   DATA[1964,13] := 797.9124;
   DATA[1964,14] := 1.0;
   DATA[1964,15] := 2.0;
   DATA[1964,16] := 1.0;
   DATA[1964,17] := 1.0;
   DATA[1964,18] := 1.0;
   DATA[1964,19] := 2.0;
   DATA[1964,20] := 148.808;
   DATA[1964,21] := 154.8065;
   DATA[1964,22] := 1.718387;
   DATA[1964,23] := 826.5958;
   DATA[1964,24] := 2.0;
   DATA[1964,25] := 2.0;
   DATA[1964,26] := 7.874455;
   DATA[1964,27] := 143.8093;
   DATA[1964,28] := 262.2084;
   DATA[1964,29] := 12.11228;
   DATA[1964,30] := 1.72725;
   DATA[1964,31] := 1.264891;
   DATA[1964,32] := 0.7352687;
   DATA[1964,33] := 0.3079781;
   DATA[1964,34] := 2.0;
   DATA[1964,35] := 250.5768;
   DATA[1964,36] := 1.730048;
   DATA[1964,37] := 189.3265;
   DATA[1964,38] := 0.000128152;
   DATA[1964,39] := 1.0;
   DATA[1964,40] := 1.0;
   DATA[1965,0] := 2.537873;
   DATA[1965,1] := 860.8522;
   DATA[1965,2] := 2.0;
   DATA[1965,3] := 2.0;
   DATA[1965,4] := 262.3686;
   DATA[1965,5] := 8.396437;
   DATA[1965,6] := 331.8893;
   DATA[1965,7] := 2.462051;
   DATA[1965,8] := 2.0;
   DATA[1965,9] := 2.0;
   DATA[1965,10] := 2.0;
   DATA[1965,11] := 19.69396;
   DATA[1965,12] := 2.209269;
   DATA[1965,13] := 797.8724;
   DATA[1965,14] := 1.0;
   DATA[1965,15] := 2.0;
   DATA[1965,16] := 1.0;
   DATA[1965,17] := 1.0;
   DATA[1965,18] := 1.0;
   DATA[1965,19] := 2.0;
   DATA[1965,20] := 148.808;
   DATA[1965,21] := 154.8065;
   DATA[1965,22] := 1.718771;
   DATA[1965,23] := 826.5189;
   DATA[1965,24] := 2.0;
   DATA[1965,25] := 2.0;
   DATA[1965,26] := 7.874455;
   DATA[1965,27] := 143.8093;
   DATA[1965,28] := 262.2084;
   DATA[1965,29] := 12.11228;
   DATA[1965,30] := 1.72725;
   DATA[1965,31] := 1.262073;
   DATA[1965,32] := 0.7352687;
   DATA[1965,33] := 0.3079781;
   DATA[1965,34] := 2.0;
   DATA[1965,35] := 250.5768;
   DATA[1965,36] := 1.730048;
   DATA[1965,37] := 189.3265;
   DATA[1965,38] := 0.000128152;
   DATA[1965,39] := 1.0;
   DATA[1965,40] := 1.0;
   DATA[1966,0] := 2.58111;
   DATA[1966,1] := 860.6559;
   DATA[1966,2] := 2.0;
   DATA[1966,3] := 2.0;
   DATA[1966,4] := 262.3686;
   DATA[1966,5] := 8.396437;
   DATA[1966,6] := 331.8893;
   DATA[1966,7] := 2.46077;
   DATA[1966,8] := 2.0;
   DATA[1966,9] := 2.0;
   DATA[1966,10] := 2.0;
   DATA[1966,11] := 19.74838;
   DATA[1966,12] := 2.21119;
   DATA[1966,13] := 797.7522;
   DATA[1966,14] := 1.0;
   DATA[1966,15] := 2.0;
   DATA[1966,16] := 1.0;
   DATA[1966,17] := 1.0;
   DATA[1966,18] := 1.0;
   DATA[1966,19] := 2.0;
   DATA[1966,20] := 148.808;
   DATA[1966,21] := 154.8065;
   DATA[1966,22] := 1.720437;
   DATA[1966,23] := 826.1728;
   DATA[1966,24] := 2.0;
   DATA[1966,25] := 2.0;
   DATA[1966,26] := 7.874455;
   DATA[1966,27] := 143.8349;
   DATA[1966,28] := 262.2084;
   DATA[1966,29] := 12.11228;
   DATA[1966,30] := 1.72725;
   DATA[1966,31] := 1.276162;
   DATA[1966,32] := 0.7352687;
   DATA[1966,33] := 0.3084905;
   DATA[1966,34] := 2.0;
   DATA[1966,35] := 250.5768;
   DATA[1966,36] := 1.730048;
   DATA[1966,37] := 189.3265;
   DATA[1966,38] := 0.000128152;
   DATA[1966,39] := 1.0;
   DATA[1966,40] := 1.0;
   DATA[1967,0] := 2.61602;
   DATA[1967,1] := 860.6167;
   DATA[1967,2] := 2.0;
   DATA[1967,3] := 2.0;
   DATA[1967,4] := 262.3686;
   DATA[1967,5] := 8.396437;
   DATA[1967,6] := 331.8893;
   DATA[1967,7] := 2.46077;
   DATA[1967,8] := 2.0;
   DATA[1967,9] := 2.0;
   DATA[1967,10] := 2.0;
   DATA[1967,11] := 19.79;
   DATA[1967,12] := 2.212343;
   DATA[1967,13] := 797.5119;
   DATA[1967,14] := 1.0;
   DATA[1967,15] := 2.0;
   DATA[1967,16] := 1.0;
   DATA[1967,17] := 1.0;
   DATA[1967,18] := 1.0;
   DATA[1967,19] := 2.0;
   DATA[1967,20] := 148.808;
   DATA[1967,21] := 154.8065;
   DATA[1967,22] := 1.721206;
   DATA[1967,23] := 826.3651;
   DATA[1967,24] := 2.0;
   DATA[1967,25] := 2.0;
   DATA[1967,26] := 7.874455;
   DATA[1967,27] := 144.0144;
   DATA[1967,28] := 262.2084;
   DATA[1967,29] := 12.11228;
   DATA[1967,30] := 1.72725;
   DATA[1967,31] := 1.289996;
   DATA[1967,32] := 0.7352687;
   DATA[1967,33] := 0.3086186;
   DATA[1967,34] := 2.0;
   DATA[1967,35] := 250.5768;
   DATA[1967,36] := 1.730048;
   DATA[1967,37] := 189.3265;
   DATA[1967,38] := 0.000128152;
   DATA[1967,39] := 1.0;
   DATA[1967,40] := 1.0;
   DATA[1968,0] := 2.6394;
   DATA[1968,1] := 860.9307;
   DATA[1968,2] := 2.0;
   DATA[1968,3] := 2.0;
   DATA[1968,4] := 262.3686;
   DATA[1968,5] := 8.396437;
   DATA[1968,6] := 331.8123;
   DATA[1968,7] := 2.46077;
   DATA[1968,8] := 2.0;
   DATA[1968,9] := 2.0;
   DATA[1968,10] := 2.0;
   DATA[1968,11] := 19.79;
   DATA[1968,12] := 2.212343;
   DATA[1968,13] := 797.7922;
   DATA[1968,14] := 1.0;
   DATA[1968,15] := 2.0;
   DATA[1968,16] := 1.0;
   DATA[1968,17] := 1.0;
   DATA[1968,18] := 1.0;
   DATA[1968,19] := 2.0;
   DATA[1968,20] := 148.808;
   DATA[1968,21] := 154.8065;
   DATA[1968,22] := 1.721206;
   DATA[1968,23] := 825.9805;
   DATA[1968,24] := 2.0;
   DATA[1968,25] := 2.0;
   DATA[1968,26] := 7.874455;
   DATA[1968,27] := 144.0144;
   DATA[1968,28] := 262.2084;
   DATA[1968,29] := 12.11228;
   DATA[1968,30] := 1.72725;
   DATA[1968,31] := 1.302933;
   DATA[1968,32] := 0.7352687;
   DATA[1968,33] := 0.3086186;
   DATA[1968,34] := 2.0;
   DATA[1968,35] := 250.5768;
   DATA[1968,36] := 1.730048;
   DATA[1968,37] := 189.3265;
   DATA[1968,38] := 0.000128152;
   DATA[1968,39] := 1.0;
   DATA[1968,40] := 1.0;
   DATA[1969,0] := 2.652532;
   DATA[1969,1] := 860.9307;
   DATA[1969,2] := 2.0;
   DATA[1969,3] := 2.0;
   DATA[1969,4] := 262.3686;
   DATA[1969,5] := 8.396437;
   DATA[1969,6] := 331.8123;
   DATA[1969,7] := 2.46077;
   DATA[1969,8] := 2.0;
   DATA[1969,9] := 2.0;
   DATA[1969,10] := 2.0;
   DATA[1969,11] := 19.79;
   DATA[1969,12] := 2.21055;
   DATA[1969,13] := 797.592;
   DATA[1969,14] := 1.0;
   DATA[1969,15] := 2.0;
   DATA[1969,16] := 1.0;
   DATA[1969,17] := 1.0;
   DATA[1969,18] := 1.0;
   DATA[1969,19] := 2.0;
   DATA[1969,20] := 148.808;
   DATA[1969,21] := 154.8065;
   DATA[1969,22] := 1.720437;
   DATA[1969,23] := 825.6345;
   DATA[1969,24] := 2.0;
   DATA[1969,25] := 2.0;
   DATA[1969,26] := 7.874455;
   DATA[1969,27] := 144.0144;
   DATA[1969,28] := 262.2084;
   DATA[1969,29] := 12.11228;
   DATA[1969,30] := 1.72725;
   DATA[1969,31] := 1.310106;
   DATA[1969,32] := 0.7352687;
   DATA[1969,33] := 0.3072735;
   DATA[1969,34] := 2.0;
   DATA[1969,35] := 250.5768;
   DATA[1969,36] := 1.730048;
   DATA[1969,37] := 189.3265;
   DATA[1969,38] := 0.000128152;
   DATA[1969,39] := 1.0;
   DATA[1969,40] := 1.0;
   DATA[1970,0] := 2.656375;
   DATA[1970,1] := 860.5382;
   DATA[1970,2] := 2.0;
   DATA[1970,3] := 2.0;
   DATA[1970,4] := 262.3686;
   DATA[1970,5] := 8.396437;
   DATA[1970,6] := 331.8123;
   DATA[1970,7] := 2.46077;
   DATA[1970,8] := 2.0;
   DATA[1970,9] := 2.0;
   DATA[1970,10] := 2.0;
   DATA[1970,11] := 19.75479;
   DATA[1970,12] := 2.209269;
   DATA[1970,13] := 797.7522;
   DATA[1970,14] := 1.0;
   DATA[1970,15] := 2.0;
   DATA[1970,16] := 1.0;
   DATA[1970,17] := 1.0;
   DATA[1970,18] := 1.0;
   DATA[1970,19] := 2.0;
   DATA[1970,20] := 148.808;
   DATA[1970,21] := 154.8065;
   DATA[1970,22] := 1.720437;
   DATA[1970,23] := 825.596;
   DATA[1970,24] := 2.0;
   DATA[1970,25] := 2.0;
   DATA[1970,26] := 7.874455;
   DATA[1970,27] := 143.8862;
   DATA[1970,28] := 262.2084;
   DATA[1970,29] := 12.11228;
   DATA[1970,30] := 1.72725;
   DATA[1970,31] := 1.302293;
   DATA[1970,32] := 0.7352687;
   DATA[1970,33] := 0.3069532;
   DATA[1970,34] := 2.0;
   DATA[1970,35] := 250.5768;
   DATA[1970,36] := 1.730048;
   DATA[1970,37] := 189.4226;
   DATA[1970,38] := 0.000128152;
   DATA[1970,39] := 1.0;
   DATA[1970,40] := 1.0;
   DATA[1971,0] := 2.639721;
   DATA[1971,1] := 860.2242;
   DATA[1971,2] := 2.0;
   DATA[1971,3] := 2.0;
   DATA[1971,4] := 262.3686;
   DATA[1971,5] := 8.396437;
   DATA[1971,6] := 331.6842;
   DATA[1971,7] := 2.461539;
   DATA[1971,8] := 2.0;
   DATA[1971,9] := 2.0;
   DATA[1971,10] := 2.0;
   DATA[1971,11] := 19.75479;
   DATA[1971,12] := 2.209013;
   DATA[1971,13] := 797.7922;
   DATA[1971,14] := 1.0;
   DATA[1971,15] := 2.0;
   DATA[1971,16] := 1.0;
   DATA[1971,17] := 1.0;
   DATA[1971,18] := 1.0;
   DATA[1971,19] := 2.0;
   DATA[1971,20] := 148.808;
   DATA[1971,21] := 154.8065;
   DATA[1971,22] := 1.720437;
   DATA[1971,23] := 826.019;
   DATA[1971,24] := 2.0;
   DATA[1971,25] := 2.0;
   DATA[1971,26] := 7.874455;
   DATA[1971,27] := 143.8862;
   DATA[1971,28] := 262.2084;
   DATA[1971,29] := 12.11228;
   DATA[1971,30] := 1.729172;
   DATA[1971,31] := 1.292814;
   DATA[1971,32] := 0.7352687;
   DATA[1971,33] := 0.3069532;
   DATA[1971,34] := 2.0;
   DATA[1971,35] := 250.5768;
   DATA[1971,36] := 1.730048;
   DATA[1971,37] := 189.4226;
   DATA[1971,38] := 0.000128152;
   DATA[1971,39] := 1.0;
   DATA[1971,40] := 1.0;
   DATA[1972,0] := 2.626909;
   DATA[1972,1] := 860.1064;
   DATA[1972,2] := 2.0;
   DATA[1972,3] := 2.0;
   DATA[1972,4] := 262.3686;
   DATA[1972,5] := 8.396437;
   DATA[1972,6] := 331.6842;
   DATA[1972,7] := 2.462564;
   DATA[1972,8] := 2.0;
   DATA[1972,9] := 2.0;
   DATA[1972,10] := 2.0;
   DATA[1972,11] := 19.71957;
   DATA[1972,12] := 2.209013;
   DATA[1972,13] := 797.6721;
   DATA[1972,14] := 1.0;
   DATA[1972,15] := 2.0;
   DATA[1972,16] := 1.0;
   DATA[1972,17] := 1.0;
   DATA[1972,18] := 1.0;
   DATA[1972,19] := 2.0;
   DATA[1972,20] := 148.808;
   DATA[1972,21] := 154.8065;
   DATA[1972,22] := 1.719796;
   DATA[1972,23] := 825.7883;
   DATA[1972,24] := 2.0;
   DATA[1972,25] := 2.0;
   DATA[1972,26] := 7.874455;
   DATA[1972,27] := 143.8862;
   DATA[1972,28] := 262.2084;
   DATA[1972,29] := 12.11228;
   DATA[1972,30] := 1.730197;
   DATA[1972,31] := 1.277956;
   DATA[1972,32] := 0.7352687;
   DATA[1972,33] := 0.3069532;
   DATA[1972,34] := 2.0;
   DATA[1972,35] := 250.5768;
   DATA[1972,36] := 1.730048;
   DATA[1972,37] := 189.4226;
   DATA[1972,38] := 0.000128152;
   DATA[1972,39] := 1.0;
   DATA[1972,40] := 1.0;
   DATA[1973,0] := 2.620184;
   DATA[1973,1] := 860.1457;
   DATA[1973,2] := 2.0;
   DATA[1973,3] := 2.0;
   DATA[1973,4] := 262.3686;
   DATA[1973,5] := 8.396437;
   DATA[1973,6] := 331.6842;
   DATA[1973,7] := 2.462564;
   DATA[1973,8] := 2.0;
   DATA[1973,9] := 2.0;
   DATA[1973,10] := 2.0;
   DATA[1973,11] := 19.70677;
   DATA[1973,12] := 2.209013;
   DATA[1973,13] := 797.6721;
   DATA[1973,14] := 1.0;
   DATA[1973,15] := 2.0;
   DATA[1973,16] := 1.0;
   DATA[1973,17] := 1.0;
   DATA[1973,18] := 1.0;
   DATA[1973,19] := 2.0;
   DATA[1973,20] := 148.808;
   DATA[1973,21] := 154.8065;
   DATA[1973,22] := 1.719796;
   DATA[1973,23] := 825.9421;
   DATA[1973,24] := 2.0;
   DATA[1973,25] := 2.0;
   DATA[1973,26] := 7.874455;
   DATA[1973,27] := 143.8862;
   DATA[1973,28] := 262.2084;
   DATA[1973,29] := 12.11228;
   DATA[1973,30] := 1.731864;
   DATA[1973,31] := 1.272192;
   DATA[1973,32] := 0.7352687;
   DATA[1973,33] := 0.3069532;
   DATA[1973,34] := 2.0;
   DATA[1973,35] := 250.5127;
   DATA[1973,36] := 1.730048;
   DATA[1973,37] := 189.4226;
   DATA[1973,38] := 0.000128152;
   DATA[1973,39] := 1.0;
   DATA[1973,40] := 1.0;
   DATA[1974,0] := 2.613778;
   DATA[1974,1] := 859.9494;
   DATA[1974,2] := 2.0;
   DATA[1974,3] := 2.0;
   DATA[1974,4] := 262.3686;
   DATA[1974,5] := 8.396437;
   DATA[1974,6] := 331.6842;
   DATA[1974,7] := 2.462564;
   DATA[1974,8] := 2.0;
   DATA[1974,9] := 2.0;
   DATA[1974,10] := 2.0;
   DATA[1974,11] := 19.68436;
   DATA[1974,12] := 2.209525;
   DATA[1974,13] := 797.7522;
   DATA[1974,14] := 1.0;
   DATA[1974,15] := 2.0;
   DATA[1974,16] := 1.0;
   DATA[1974,17] := 1.0;
   DATA[1974,18] := 1.0;
   DATA[1974,19] := 2.0;
   DATA[1974,20] := 148.808;
   DATA[1974,21] := 154.8065;
   DATA[1974,22] := 1.71813;
   DATA[1974,23] := 826.1343;
   DATA[1974,24] := 2.0;
   DATA[1974,25] := 2.0;
   DATA[1974,26] := 7.874455;
   DATA[1974,27] := 143.8862;
   DATA[1974,28] := 262.2084;
   DATA[1974,29] := 12.11228;
   DATA[1974,30] := 1.731864;
   DATA[1974,31] := 1.265147;
   DATA[1974,32] := 0.7352687;
   DATA[1974,33] := 0.3069532;
   DATA[1974,34] := 2.0;
   DATA[1974,35] := 250.5127;
   DATA[1974,36] := 1.730048;
   DATA[1974,37] := 189.4226;
   DATA[1974,38] := 0.000128152;
   DATA[1974,39] := 1.0;
   DATA[1974,40] := 1.0;
   DATA[1975,0] := 2.601608;
   DATA[1975,1] := 859.8709;
   DATA[1975,2] := 2.0;
   DATA[1975,3] := 2.0;
   DATA[1975,4] := 262.3686;
   DATA[1975,5] := 8.396437;
   DATA[1975,6] := 331.6842;
   DATA[1975,7] := 2.462564;
   DATA[1975,8] := 2.0;
   DATA[1975,9] := 2.0;
   DATA[1975,10] := 2.0;
   DATA[1975,11] := 19.66195;
   DATA[1975,12] := 2.209525;
   DATA[1975,13] := 797.9925;
   DATA[1975,14] := 1.0;
   DATA[1975,15] := 2.0;
   DATA[1975,16] := 1.0;
   DATA[1975,17] := 1.0;
   DATA[1975,18] := 1.0;
   DATA[1975,19] := 2.0;
   DATA[1975,20] := 148.808;
   DATA[1975,21] := 154.8065;
   DATA[1975,22] := 1.71813;
   DATA[1975,23] := 826.442;
   DATA[1975,24] := 2.0;
   DATA[1975,25] := 2.0;
   DATA[1975,26] := 7.874455;
   DATA[1975,27] := 143.8862;
   DATA[1975,28] := 262.2084;
   DATA[1975,29] := 12.11228;
   DATA[1975,30] := 1.731095;
   DATA[1975,31] := 1.26425;
   DATA[1975,32] := 0.7352687;
   DATA[1975,33] := 0.3066329;
   DATA[1975,34] := 2.0;
   DATA[1975,35] := 250.5127;
   DATA[1975,36] := 1.730048;
   DATA[1975,37] := 189.4226;
   DATA[1975,38] := 0.000128152;
   DATA[1975,39] := 1.0;
   DATA[1975,40] := 1.0;
   DATA[1976,0] := 2.583352;
   DATA[1976,1] := 859.7139;
   DATA[1976,2] := 2.0;
   DATA[1976,3] := 2.0;
   DATA[1976,4] := 262.3686;
   DATA[1976,5] := 8.396437;
   DATA[1976,6] := 331.6842;
   DATA[1976,7] := 2.462564;
   DATA[1976,8] := 2.0;
   DATA[1976,9] := 2.0;
   DATA[1976,10] := 2.0;
   DATA[1976,11] := 19.66195;
   DATA[1976,12] := 2.209525;
   DATA[1976,13] := 797.9925;
   DATA[1976,14] := 1.0;
   DATA[1976,15] := 2.0;
   DATA[1976,16] := 1.0;
   DATA[1976,17] := 1.0;
   DATA[1976,18] := 1.0;
   DATA[1976,19] := 2.0;
   DATA[1976,20] := 148.808;
   DATA[1976,21] := 154.8065;
   DATA[1976,22] := 1.71813;
   DATA[1976,23] := 826.5189;
   DATA[1976,24] := 2.0;
   DATA[1976,25] := 2.0;
   DATA[1976,26] := 7.874455;
   DATA[1976,27] := 143.8862;
   DATA[1976,28] := 262.2084;
   DATA[1976,29] := 12.03538;
   DATA[1976,30] := 1.731095;
   DATA[1976,31] := 1.271935;
   DATA[1976,32] := 0.7352687;
   DATA[1976,33] := 0.3065048;
   DATA[1976,34] := 2.0;
   DATA[1976,35] := 250.5127;
   DATA[1976,36] := 1.730048;
   DATA[1976,37] := 189.4226;
   DATA[1976,38] := 0.000128152;
   DATA[1976,39] := 1.0;
   DATA[1976,40] := 1.0;
   DATA[1977,0] := 2.572463;
   DATA[1977,1] := 859.8317;
   DATA[1977,2] := 2.0;
   DATA[1977,3] := 2.0;
   DATA[1977,4] := 262.3686;
   DATA[1977,5] := 8.396437;
   DATA[1977,6] := 331.6842;
   DATA[1977,7] := 2.462564;
   DATA[1977,8] := 2.0;
   DATA[1977,9] := 2.0;
   DATA[1977,10] := 2.0;
   DATA[1977,11] := 19.70037;
   DATA[1977,12] := 2.209525;
   DATA[1977,13] := 798.353;
   DATA[1977,14] := 1.0;
   DATA[1977,15] := 2.0;
   DATA[1977,16] := 1.0;
   DATA[1977,17] := 1.0;
   DATA[1977,18] := 1.0;
   DATA[1977,19] := 2.0;
   DATA[1977,20] := 148.808;
   DATA[1977,21] := 154.8065;
   DATA[1977,22] := 1.71813;
   DATA[1977,23] := 826.5573;
   DATA[1977,24] := 2.0;
   DATA[1977,25] := 2.0;
   DATA[1977,26] := 7.874455;
   DATA[1977,27] := 143.8862;
   DATA[1977,28] := 262.2084;
   DATA[1977,29] := 12.03538;
   DATA[1977,30] := 1.731095;
   DATA[1977,31] := 1.271935;
   DATA[1977,32] := 0.7352687;
   DATA[1977,33] := 0.3065048;
   DATA[1977,34] := 2.0;
   DATA[1977,35] := 250.5127;
   DATA[1977,36] := 1.730048;
   DATA[1977,37] := 189.2464;
   DATA[1977,38] := 0.000128152;
   DATA[1977,39] := 1.0;
   DATA[1977,40] := 1.0;
   DATA[1978,0] := 2.556769;
   DATA[1978,1] := 859.6354;
   DATA[1978,2] := 2.0;
   DATA[1978,3] := 2.0;
   DATA[1978,4] := 262.3686;
   DATA[1978,5] := 8.396437;
   DATA[1978,6] := 331.6842;
   DATA[1978,7] := 2.462564;
   DATA[1978,8] := 2.0;
   DATA[1978,9] := 2.0;
   DATA[1978,10] := 2.0;
   DATA[1978,11] := 19.76439;
   DATA[1978,12] := 2.209525;
   DATA[1978,13] := 798.7535;
   DATA[1978,14] := 1.0;
   DATA[1978,15] := 2.0;
   DATA[1978,16] := 1.0;
   DATA[1978,17] := 1.0;
   DATA[1978,18] := 1.0;
   DATA[1978,19] := 2.0;
   DATA[1978,20] := 148.808;
   DATA[1978,21] := 154.8065;
   DATA[1978,22] := 1.716721;
   DATA[1978,23] := 826.6342;
   DATA[1978,24] := 2.0;
   DATA[1978,25] := 2.0;
   DATA[1978,26] := 7.874455;
   DATA[1978,27] := 143.8862;
   DATA[1978,28] := 262.2084;
   DATA[1978,29] := 12.03538;
   DATA[1978,30] := 1.7293;
   DATA[1978,31] := 1.280517;
   DATA[1978,32] := 0.7352687;
   DATA[1978,33] := 0.3065048;
   DATA[1978,34] := 2.0;
   DATA[1978,35] := 250.5127;
   DATA[1978,36] := 1.730048;
   DATA[1978,37] := 189.2464;
   DATA[1978,38] := 0.000128152;
   DATA[1978,39] := 1.0;
   DATA[1978,40] := 1.0;
   DATA[1979,0] := 2.53435;
   DATA[1979,1] := 859.9494;
   DATA[1979,2] := 2.0;
   DATA[1979,3] := 2.0;
   DATA[1979,4] := 262.3686;
   DATA[1979,5] := 8.396437;
   DATA[1979,6] := 331.6842;
   DATA[1979,7] := 2.462564;
   DATA[1979,8] := 2.0;
   DATA[1979,9] := 2.0;
   DATA[1979,10] := 2.0;
   DATA[1979,11] := 19.76439;
   DATA[1979,12] := 2.209525;
   DATA[1979,13] := 798.6735;
   DATA[1979,14] := 1.0;
   DATA[1979,15] := 2.0;
   DATA[1979,16] := 1.0;
   DATA[1979,17] := 1.0;
   DATA[1979,18] := 1.0;
   DATA[1979,19] := 2.0;
   DATA[1979,20] := 148.808;
   DATA[1979,21] := 154.8065;
   DATA[1979,22] := 1.716721;
   DATA[1979,23] := 826.3266;
   DATA[1979,24] := 2.0;
   DATA[1979,25] := 2.0;
   DATA[1979,26] := 7.874455;
   DATA[1979,27] := 143.8862;
   DATA[1979,28] := 262.2084;
   DATA[1979,29] := 12.03538;
   DATA[1979,30] := 1.728147;
   DATA[1979,31] := 1.280902;
   DATA[1979,32] := 0.7352687;
   DATA[1979,33] := 0.3065048;
   DATA[1979,34] := 2.0;
   DATA[1979,35] := 250.5127;
   DATA[1979,36] := 1.730048;
   DATA[1979,37] := 189.2464;
   DATA[1979,38] := 0.000128152;
   DATA[1979,39] := 1.0;
   DATA[1979,40] := 1.0;
   DATA[1980,0] := 2.518015;
   DATA[1980,1] := 859.6354;
   DATA[1980,2] := 2.0;
   DATA[1980,3] := 2.0;
   DATA[1980,4] := 262.3686;
   DATA[1980,5] := 8.396437;
   DATA[1980,6] := 331.6842;
   DATA[1980,7] := 2.462564;
   DATA[1980,8] := 2.0;
   DATA[1980,9] := 2.0;
   DATA[1980,10] := 2.0;
   DATA[1980,11] := 19.7996;
   DATA[1980,12] := 2.209525;
   DATA[1980,13] := 799.074;
   DATA[1980,14] := 1.0;
   DATA[1980,15] := 2.0;
   DATA[1980,16] := 1.0;
   DATA[1980,17] := 1.0;
   DATA[1980,18] := 1.0;
   DATA[1980,19] := 2.0;
   DATA[1980,20] := 148.808;
   DATA[1980,21] := 155.0372;
   DATA[1980,22] := 1.716721;
   DATA[1980,23] := 826.8265;
   DATA[1980,24] := 2.0;
   DATA[1980,25] := 2.0;
   DATA[1980,26] := 7.874455;
   DATA[1980,27] := 143.8862;
   DATA[1980,28] := 262.2084;
   DATA[1980,29] := 12.03538;
   DATA[1980,30] := 1.726865;
   DATA[1980,31] := 1.271679;
   DATA[1980,32] := 0.7352687;
   DATA[1980,33] := 0.3065048;
   DATA[1980,34] := 2.0;
   DATA[1980,35] := 250.5127;
   DATA[1980,36] := 1.730048;
   DATA[1980,37] := 189.3745;
   DATA[1980,38] := 0.000128152;
   DATA[1980,39] := 1.0;
   DATA[1980,40] := 1.0;
   DATA[1981,0] := 2.499439;
   DATA[1981,1] := 859.4391;
   DATA[1981,2] := 2.0;
   DATA[1981,3] := 2.0;
   DATA[1981,4] := 262.3686;
   DATA[1981,5] := 8.396437;
   DATA[1981,6] := 331.6842;
   DATA[1981,7] := 2.462564;
   DATA[1981,8] := 2.0;
   DATA[1981,9] := 2.0;
   DATA[1981,10] := 2.0;
   DATA[1981,11] := 19.7996;
   DATA[1981,12] := 2.209525;
   DATA[1981,13] := 799.3143;
   DATA[1981,14] := 1.0;
   DATA[1981,15] := 2.0;
   DATA[1981,16] := 1.0;
   DATA[1981,17] := 1.0;
   DATA[1981,18] := 1.0;
   DATA[1981,19] := 2.0;
   DATA[1981,20] := 148.808;
   DATA[1981,21] := 155.0372;
   DATA[1981,22] := 1.716721;
   DATA[1981,23] := 826.7496;
   DATA[1981,24] := 2.0;
   DATA[1981,25] := 2.0;
   DATA[1981,26] := 7.874455;
   DATA[1981,27] := 143.8862;
   DATA[1981,28] := 262.2084;
   DATA[1981,29] := 12.03538;
   DATA[1981,30] := 1.726865;
   DATA[1981,31] := 1.275394;
   DATA[1981,32] := 0.7352687;
   DATA[1981,33] := 0.3065048;
   DATA[1981,34] := 2.0;
   DATA[1981,35] := 250.5127;
   DATA[1981,36] := 1.730048;
   DATA[1981,37] := 189.4066;
   DATA[1981,38] := 0.000128152;
   DATA[1981,39] := 1.0;
   DATA[1981,40] := 1.0;
   DATA[1982,0] := 2.482465;
   DATA[1982,1] := 859.3214;
   DATA[1982,2] := 2.0;
   DATA[1982,3] := 2.0;
   DATA[1982,4] := 262.3686;
   DATA[1982,5] := 8.396437;
   DATA[1982,6] := 331.5047;
   DATA[1982,7] := 2.462307;
   DATA[1982,8] := 2.0;
   DATA[1982,9] := 2.0;
   DATA[1982,10] := 2.0;
   DATA[1982,11] := 19.71957;
   DATA[1982,12] := 2.209525;
   DATA[1982,13] := 799.1942;
   DATA[1982,14] := 1.0;
   DATA[1982,15] := 2.0;
   DATA[1982,16] := 1.0;
   DATA[1982,17] := 1.0;
   DATA[1982,18] := 1.0;
   DATA[1982,19] := 2.0;
   DATA[1982,20] := 148.808;
   DATA[1982,21] := 155.0372;
   DATA[1982,22] := 1.716721;
   DATA[1982,23] := 827.3264;
   DATA[1982,24] := 2.0;
   DATA[1982,25] := 2.0;
   DATA[1982,26] := 7.874455;
   DATA[1982,27] := 143.8862;
   DATA[1982,28] := 262.2084;
   DATA[1982,29] := 12.03538;
   DATA[1982,30] := 1.726865;
   DATA[1982,31] := 1.296273;
   DATA[1982,32] := 0.7352687;
   DATA[1982,33] := 0.3065048;
   DATA[1982,34] := 2.0;
   DATA[1982,35] := 250.5127;
   DATA[1982,36] := 1.730048;
   DATA[1982,37] := 189.4066;
   DATA[1982,38] := 0.000128152;
   DATA[1982,39] := 1.0;
   DATA[1982,40] := 1.0;
   DATA[1983,0] := 2.462287;
   DATA[1983,1] := 859.3607;
   DATA[1983,2] := 2.0;
   DATA[1983,3] := 2.0;
   DATA[1983,4] := 262.3686;
   DATA[1983,5] := 8.396437;
   DATA[1983,6] := 331.5047;
   DATA[1983,7] := 2.462307;
   DATA[1983,8] := 2.0;
   DATA[1983,9] := 2.0;
   DATA[1983,10] := 2.0;
   DATA[1983,11] := 19.71957;
   DATA[1983,12] := 2.209525;
   DATA[1983,13] := 799.9551;
   DATA[1983,14] := 1.0;
   DATA[1983,15] := 2.0;
   DATA[1983,16] := 1.0;
   DATA[1983,17] := 1.0;
   DATA[1983,18] := 1.0;
   DATA[1983,19] := 2.0;
   DATA[1983,20] := 148.808;
   DATA[1983,21] := 154.8834;
   DATA[1983,22] := 1.716721;
   DATA[1983,23] := 826.9418;
   DATA[1983,24] := 2.0;
   DATA[1983,25] := 2.0;
   DATA[1983,26] := 7.874455;
   DATA[1983,27] := 143.6298;
   DATA[1983,28] := 262.2084;
   DATA[1983,29] := 12.03538;
   DATA[1983,30] := 1.726865;
   DATA[1983,31] := 1.302677;
   DATA[1983,32] := 0.7352687;
   DATA[1983,33] := 0.3065048;
   DATA[1983,34] := 2.0;
   DATA[1983,35] := 250.5127;
   DATA[1983,36] := 1.730048;
   DATA[1983,37] := 189.4066;
   DATA[1983,38] := 0.000128152;
   DATA[1983,39] := 1.0;
   DATA[1983,40] := 1.0;
   DATA[1984,0] := 2.451398;
   DATA[1984,1] := 859.5176;
   DATA[1984,2] := 2.0;
   DATA[1984,3] := 2.0;
   DATA[1984,4] := 262.3686;
   DATA[1984,5] := 8.396437;
   DATA[1984,6] := 331.5047;
   DATA[1984,7] := 2.462307;
   DATA[1984,8] := 2.0;
   DATA[1984,9] := 2.0;
   DATA[1984,10] := 2.0;
   DATA[1984,11] := 19.71957;
   DATA[1984,12] := 2.209525;
   DATA[1984,13] := 800.1955;
   DATA[1984,14] := 1.0;
   DATA[1984,15] := 2.0;
   DATA[1984,16] := 1.0;
   DATA[1984,17] := 1.0;
   DATA[1984,18] := 1.0;
   DATA[1984,19] := 2.0;
   DATA[1984,20] := 148.808;
   DATA[1984,21] := 154.8834;
   DATA[1984,22] := 1.716721;
   DATA[1984,23] := 826.9803;
   DATA[1984,24] := 2.0;
   DATA[1984,25] := 2.0;
   DATA[1984,26] := 7.874455;
   DATA[1984,27] := 143.6298;
   DATA[1984,28] := 262.2084;
   DATA[1984,29] := 12.03538;
   DATA[1984,30] := 1.726865;
   DATA[1984,31] := 1.311259;
   DATA[1984,32] := 0.7352687;
   DATA[1984,33] := 0.3065048;
   DATA[1984,34] := 2.0;
   DATA[1984,35] := 250.5127;
   DATA[1984,36] := 1.730048;
   DATA[1984,37] := 189.4066;
   DATA[1984,38] := 0.000128152;
   DATA[1984,39] := 1.0;
   DATA[1984,40] := 1.0;
   DATA[1985,0] := 2.433783;
   DATA[1985,1] := 859.9102;
   DATA[1985,2] := 2.0;
   DATA[1985,3] := 2.0;
   DATA[1985,4] := 262.3686;
   DATA[1985,5] := 8.396437;
   DATA[1985,6] := 331.4535;
   DATA[1985,7] := 2.462307;
   DATA[1985,8] := 2.0;
   DATA[1985,9] := 2.0;
   DATA[1985,10] := 2.0;
   DATA[1985,11] := 19.73238;
   DATA[1985,12] := 2.209525;
   DATA[1985,13] := 800.556;
   DATA[1985,14] := 1.0;
   DATA[1985,15] := 2.0;
   DATA[1985,16] := 1.0;
   DATA[1985,17] := 1.0;
   DATA[1985,18] := 1.0;
   DATA[1985,19] := 2.0;
   DATA[1985,20] := 148.808;
   DATA[1985,21] := 154.8834;
   DATA[1985,22] := 1.719156;
   DATA[1985,23] := 826.442;
   DATA[1985,24] := 2.0;
   DATA[1985,25] := 2.0;
   DATA[1985,26] := 7.874455;
   DATA[1985,27] := 143.6298;
   DATA[1985,28] := 262.0802;
   DATA[1985,29] := 12.30454;
   DATA[1985,30] := 1.728147;
   DATA[1985,31] := 1.306648;
   DATA[1985,32] := 0.7352687;
   DATA[1985,33] := 0.3065048;
   DATA[1985,34] := 2.0;
   DATA[1985,35] := 250.5127;
   DATA[1985,36] := 1.730048;
   DATA[1985,37] := 189.4066;
   DATA[1985,38] := 0.000128152;
   DATA[1985,39] := 1.0;
   DATA[1985,40] := 1.0;
   DATA[1986,0] := 2.428338;
   DATA[1986,1] := 859.9102;
   DATA[1986,2] := 2.0;
   DATA[1986,3] := 2.0;
   DATA[1986,4] := 262.3686;
   DATA[1986,5] := 8.396437;
   DATA[1986,6] := 331.4535;
   DATA[1986,7] := 2.461923;
   DATA[1986,8] := 2.0;
   DATA[1986,9] := 2.0;
   DATA[1986,10] := 2.0;
   DATA[1986,11] := 19.7804;
   DATA[1986,12] := 2.209525;
   DATA[1986,13] := 801.1568;
   DATA[1986,14] := 1.0;
   DATA[1986,15] := 2.0;
   DATA[1986,16] := 1.0;
   DATA[1986,17] := 1.0;
   DATA[1986,18] := 1.0;
   DATA[1986,19] := 2.0;
   DATA[1986,20] := 148.808;
   DATA[1986,21] := 154.8834;
   DATA[1986,22] := 1.719156;
   DATA[1986,23] := 826.8265;
   DATA[1986,24] := 2.0;
   DATA[1986,25] := 2.0;
   DATA[1986,26] := 7.874455;
   DATA[1986,27] := 143.6298;
   DATA[1986,28] := 262.0802;
   DATA[1986,29] := 12.30454;
   DATA[1986,30] := 1.7293;
   DATA[1986,31] := 1.301396;
   DATA[1986,32] := 0.7352687;
   DATA[1986,33] := 0.3065048;
   DATA[1986,34] := 2.0;
   DATA[1986,35] := 250.5127;
   DATA[1986,36] := 1.730048;
   DATA[1986,37] := 189.4066;
   DATA[1986,38] := 0.000128152;
   DATA[1986,39] := 1.0;
   DATA[1986,40] := 1.0;
   DATA[1987,0] := 2.428018;
   DATA[1987,1] := 859.9494;
   DATA[1987,2] := 2.0;
   DATA[1987,3] := 2.0;
   DATA[1987,4] := 262.3686;
   DATA[1987,5] := 8.392271;
   DATA[1987,6] := 331.4535;
   DATA[1987,7] := 2.461923;
   DATA[1987,8] := 2.0;
   DATA[1987,9] := 2.0;
   DATA[1987,10] := 2.0;
   DATA[1987,11] := 19.73558;
   DATA[1987,12] := 2.209525;
   DATA[1987,13] := 800.9966;
   DATA[1987,14] := 1.0;
   DATA[1987,15] := 2.0;
   DATA[1987,16] := 1.0;
   DATA[1987,17] := 1.0;
   DATA[1987,18] := 1.0;
   DATA[1987,19] := 2.0;
   DATA[1987,20] := 148.808;
   DATA[1987,21] := 154.8834;
   DATA[1987,22] := 1.717233;
   DATA[1987,23] := 826.4035;
   DATA[1987,24] := 2.0;
   DATA[1987,25] := 2.0;
   DATA[1987,26] := 7.874455;
   DATA[1987,27] := 143.6298;
   DATA[1987,28] := 262.0802;
   DATA[1987,29] := 12.26609;
   DATA[1987,30] := 1.729428;
   DATA[1987,31] := 1.30716;
   DATA[1987,32] := 0.7352687;
   DATA[1987,33] := 0.3065048;
   DATA[1987,34] := 2.0;
   DATA[1987,35] := 250.5127;
   DATA[1987,36] := 1.730048;
   DATA[1987,37] := 189.4066;
   DATA[1987,38] := 0.000128152;
   DATA[1987,39] := 1.0;
   DATA[1987,40] := 1.0;
   DATA[1988,0] := 2.428018;
   DATA[1988,1] := 859.8317;
   DATA[1988,2] := 2.0;
   DATA[1988,3] := 2.0;
   DATA[1988,4] := 262.3686;
   DATA[1988,5] := 8.392271;
   DATA[1988,6] := 331.4535;
   DATA[1988,7] := 2.461923;
   DATA[1988,8] := 2.0;
   DATA[1988,9] := 2.0;
   DATA[1988,10] := 2.0;
   DATA[1988,11] := 19.73558;
   DATA[1988,12] := 2.209525;
   DATA[1988,13] := 801.5173;
   DATA[1988,14] := 1.0;
   DATA[1988,15] := 2.0;
   DATA[1988,16] := 1.0;
   DATA[1988,17] := 1.0;
   DATA[1988,18] := 1.0;
   DATA[1988,19] := 2.0;
   DATA[1988,20] := 148.808;
   DATA[1988,21] := 154.8834;
   DATA[1988,22] := 1.714798;
   DATA[1988,23] := 826.5189;
   DATA[1988,24] := 2.0;
   DATA[1988,25] := 2.0;
   DATA[1988,26] := 7.874455;
   DATA[1988,27] := 143.6298;
   DATA[1988,28] := 262.0802;
   DATA[1988,29] := 11.88157;
   DATA[1988,30] := 1.729428;
   DATA[1988,31] := 1.320994;
   DATA[1988,32] := 0.7352687;
   DATA[1988,33] := 0.3065048;
   DATA[1988,34] := 2.0;
   DATA[1988,35] := 250.5127;
   DATA[1988,36] := 1.730048;
   DATA[1988,37] := 189.4066;
   DATA[1988,38] := 0.000128152;
   DATA[1988,39] := 1.0;
   DATA[1988,40] := 1.0;
   DATA[1989,0] := 2.472216;
   DATA[1989,1] := 859.8709;
   DATA[1989,2] := 2.0;
   DATA[1989,3] := 2.0;
   DATA[1989,4] := 262.3686;
   DATA[1989,5] := 8.392271;
   DATA[1989,6] := 331.4535;
   DATA[1989,7] := 2.463204;
   DATA[1989,8] := 2.0;
   DATA[1989,9] := 2.0;
   DATA[1989,10] := 2.0;
   DATA[1989,11] := 19.73558;
   DATA[1989,12] := 2.209525;
   DATA[1989,13] := 801.317;
   DATA[1989,14] := 1.0;
   DATA[1989,15] := 2.0;
   DATA[1989,16] := 1.0;
   DATA[1989,17] := 1.0;
   DATA[1989,18] := 1.0;
   DATA[1989,19] := 2.0;
   DATA[1989,20] := 148.808;
   DATA[1989,21] := 154.8834;
   DATA[1989,22] := 1.714798;
   DATA[1989,23] := 826.7111;
   DATA[1989,24] := 2.0;
   DATA[1989,25] := 2.0;
   DATA[1989,26] := 7.874455;
   DATA[1989,27] := 143.6298;
   DATA[1989,28] := 262.0802;
   DATA[1989,29] := 11.88157;
   DATA[1989,30] := 1.729428;
   DATA[1989,31] := 1.321634;
   DATA[1989,32] := 0.7352687;
   DATA[1989,33] := 0.3065048;
   DATA[1989,34] := 2.0;
   DATA[1989,35] := 250.5127;
   DATA[1989,36] := 1.730048;
   DATA[1989,37] := 189.4066;
   DATA[1989,38] := 0.000128152;
   DATA[1989,39] := 1.0;
   DATA[1989,40] := 1.0;
   DATA[1990,0] := 2.526022;
   DATA[1990,1] := 859.8317;
   DATA[1990,2] := 2.0;
   DATA[1990,3] := 2.0;
   DATA[1990,4] := 262.3686;
   DATA[1990,5] := 8.392271;
   DATA[1990,6] := 331.4535;
   DATA[1990,7] := 2.464742;
   DATA[1990,8] := 2.0;
   DATA[1990,9] := 2.0;
   DATA[1990,10] := 2.0;
   DATA[1990,11] := 19.73558;
   DATA[1990,12] := 2.209525;
   DATA[1990,13] := 801.317;
   DATA[1990,14] := 1.0;
   DATA[1990,15] := 2.0;
   DATA[1990,16] := 1.0;
   DATA[1990,17] := 1.0;
   DATA[1990,18] := 1.0;
   DATA[1990,19] := 2.0;
   DATA[1990,20] := 148.808;
   DATA[1990,21] := 154.8834;
   DATA[1990,22] := 1.714798;
   DATA[1990,23] := 826.788;
   DATA[1990,24] := 2.0;
   DATA[1990,25] := 2.0;
   DATA[1990,26] := 7.874455;
   DATA[1990,27] := 143.6298;
   DATA[1990,28] := 262.0802;
   DATA[1990,29] := 11.88157;
   DATA[1990,30] := 1.729428;
   DATA[1990,31] := 1.315614;
   DATA[1990,32] := 0.7352687;
   DATA[1990,33] := 0.3065048;
   DATA[1990,34] := 2.0;
   DATA[1990,35] := 250.5768;
   DATA[1990,36] := 1.730048;
   DATA[1990,37] := 189.4066;
   DATA[1990,38] := 0.000128152;
   DATA[1990,39] := 1.0;
   DATA[1990,40] := 1.0;
   DATA[1991,0] := 2.578548;
   DATA[1991,1] := 859.8317;
   DATA[1991,2] := 2.0;
   DATA[1991,3] := 2.0;
   DATA[1991,4] := 262.3686;
   DATA[1991,5] := 8.392271;
   DATA[1991,6] := 331.4535;
   DATA[1991,7] := 2.464742;
   DATA[1991,8] := 2.0;
   DATA[1991,9] := 2.0;
   DATA[1991,10] := 2.0;
   DATA[1991,11] := 19.73558;
   DATA[1991,12] := 2.209525;
   DATA[1991,13] := 801.6775;
   DATA[1991,14] := 1.0;
   DATA[1991,15] := 2.0;
   DATA[1991,16] := 1.0;
   DATA[1991,17] := 1.0;
   DATA[1991,18] := 1.0;
   DATA[1991,19] := 2.0;
   DATA[1991,20] := 148.808;
   DATA[1991,21] := 154.8834;
   DATA[1991,22] := 1.714286;
   DATA[1991,23] := 827.1341;
   DATA[1991,24] := 2.0;
   DATA[1991,25] := 2.0;
   DATA[1991,26] := 7.874455;
   DATA[1991,27] := 143.6298;
   DATA[1991,28] := 262.0802;
   DATA[1991,29] := 12.07383;
   DATA[1991,30] := 1.729428;
   DATA[1991,31] := 1.295376;
   DATA[1991,32] := 0.7352687;
   DATA[1991,33] := 0.3065048;
   DATA[1991,34] := 2.0;
   DATA[1991,35] := 250.5768;
   DATA[1991,36] := 1.730048;
   DATA[1991,37] := 189.4066;
   DATA[1991,38] := 0.000128152;
   DATA[1991,39] := 1.0;
   DATA[1991,40] := 1.0;
   DATA[1992,0] := 2.608974;
   DATA[1992,1] := 860.2634;
   DATA[1992,2] := 2.0;
   DATA[1992,3] := 2.0;
   DATA[1992,4] := 262.3686;
   DATA[1992,5] := 8.392271;
   DATA[1992,6] := 331.4535;
   DATA[1992,7] := 2.46282;
   DATA[1992,8] := 2.0;
   DATA[1992,9] := 2.0;
   DATA[1992,10] := 2.0;
   DATA[1992,11] := 19.73558;
   DATA[1992,12] := 2.209525;
   DATA[1992,13] := 801.5573;
   DATA[1992,14] := 1.0;
   DATA[1992,15] := 2.0;
   DATA[1992,16] := 1.0;
   DATA[1992,17] := 1.0;
   DATA[1992,18] := 1.0;
   DATA[1992,19] := 2.0;
   DATA[1992,20] := 148.808;
   DATA[1992,21] := 154.8834;
   DATA[1992,22] := 1.713004;
   DATA[1992,23] := 826.9418;
   DATA[1992,24] := 2.0;
   DATA[1992,25] := 2.0;
   DATA[1992,26] := 7.874455;
   DATA[1992,27] := 143.6298;
   DATA[1992,28] := 262.0802;
   DATA[1992,29] := 12.07383;
   DATA[1992,30] := 1.729172;
   DATA[1992,31] := 1.299091;
   DATA[1992,32] := 0.7352687;
   DATA[1992,33] := 0.3065048;
   DATA[1992,34] := 2.0;
   DATA[1992,35] := 250.6569;
   DATA[1992,36] := 1.730048;
   DATA[1992,37] := 189.4066;
   DATA[1992,38] := 0.000128152;
   DATA[1992,39] := 1.0;
   DATA[1992,40] := 1.0;
   DATA[1993,0] := 2.633635;
   DATA[1993,1] := 860.4205;
   DATA[1993,2] := 2.0;
   DATA[1993,3] := 2.0;
   DATA[1993,4] := 262.3686;
   DATA[1993,5] := 8.392271;
   DATA[1993,6] := 331.4535;
   DATA[1993,7] := 2.46282;
   DATA[1993,8] := 2.0;
   DATA[1993,9] := 2.0;
   DATA[1993,10] := 2.0;
   DATA[1993,11] := 19.73558;
   DATA[1993,12] := 2.209525;
   DATA[1993,13] := 801.7175;
   DATA[1993,14] := 1.0;
   DATA[1993,15] := 2.0;
   DATA[1993,16] := 1.0;
   DATA[1993,17] := 1.0;
   DATA[1993,18] := 1.0;
   DATA[1993,19] := 2.0;
   DATA[1993,20] := 148.808;
   DATA[1993,21] := 154.8834;
   DATA[1993,22] := 1.713004;
   DATA[1993,23] := 827.0956;
   DATA[1993,24] := 2.0;
   DATA[1993,25] := 2.0;
   DATA[1993,26] := 7.874455;
   DATA[1993,27] := 143.9375;
   DATA[1993,28] := 262.0802;
   DATA[1993,29] := 12.07383;
   DATA[1993,30] := 1.728788;
   DATA[1993,31] := 1.302037;
   DATA[1993,32] := 0.7352687;
   DATA[1993,33] := 0.3065048;
   DATA[1993,34] := 2.0;
   DATA[1993,35] := 250.721;
   DATA[1993,36] := 1.730048;
   DATA[1993,37] := 189.4066;
   DATA[1993,38] := 0.000128152;
   DATA[1993,39] := 1.0;
   DATA[1993,40] := 1.0;
   DATA[1994,0] := 2.643564;
   DATA[1994,1] := 861.0093;
   DATA[1994,2] := 2.0;
   DATA[1994,3] := 2.0;
   DATA[1994,4] := 262.3686;
   DATA[1994,5] := 8.392271;
   DATA[1994,6] := 331.4535;
   DATA[1994,7] := 2.46282;
   DATA[1994,8] := 2.0;
   DATA[1994,9] := 2.0;
   DATA[1994,10] := 2.0;
   DATA[1994,11] := 19.66195;
   DATA[1994,12] := 2.209525;
   DATA[1994,13] := 801.9578;
   DATA[1994,14] := 1.0;
   DATA[1994,15] := 2.0;
   DATA[1994,16] := 1.0;
   DATA[1994,17] := 1.0;
   DATA[1994,18] := 1.0;
   DATA[1994,19] := 2.0;
   DATA[1994,20] := 148.808;
   DATA[1994,21] := 154.8834;
   DATA[1994,22] := 1.715311;
   DATA[1994,23] := 826.9418;
   DATA[1994,24] := 2.0;
   DATA[1994,25] := 2.0;
   DATA[1994,26] := 7.874455;
   DATA[1994,27] := 143.9375;
   DATA[1994,28] := 262.0802;
   DATA[1994,29] := 12.07383;
   DATA[1994,30] := 1.728531;
   DATA[1994,31] := 1.312284;
   DATA[1994,32] := 0.7352687;
   DATA[1994,33] := 0.3065048;
   DATA[1994,34] := 2.0;
   DATA[1994,35] := 250.721;
   DATA[1994,36] := 1.730048;
   DATA[1994,37] := 189.5187;
   DATA[1994,38] := 0.000128152;
   DATA[1994,39] := 1.0;
   DATA[1994,40] := 1.0;
   DATA[1995,0] := 2.644525;
   DATA[1995,1] := 860.9307;
   DATA[1995,2] := 2.0;
   DATA[1995,3] := 2.0;
   DATA[1995,4] := 262.3686;
   DATA[1995,5] := 8.392271;
   DATA[1995,6] := 331.4535;
   DATA[1995,7] := 2.46282;
   DATA[1995,8] := 2.0;
   DATA[1995,9] := 2.0;
   DATA[1995,10] := 2.0;
   DATA[1995,11] := 19.63634;
   DATA[1995,12] := 2.209525;
   DATA[1995,13] := 801.9578;
   DATA[1995,14] := 1.0;
   DATA[1995,15] := 2.0;
   DATA[1995,16] := 1.0;
   DATA[1995,17] := 1.0;
   DATA[1995,18] := 1.0;
   DATA[1995,19] := 2.0;
   DATA[1995,20] := 148.808;
   DATA[1995,21] := 154.8834;
   DATA[1995,22] := 1.716721;
   DATA[1995,23] := 827.3264;
   DATA[1995,24] := 2.0;
   DATA[1995,25] := 2.0;
   DATA[1995,26] := 7.874455;
   DATA[1995,27] := 143.9375;
   DATA[1995,28] := 262.0802;
   DATA[1995,29] := 12.07383;
   DATA[1995,30] := 1.728531;
   DATA[1995,31] := 1.312284;
   DATA[1995,32] := 0.7352687;
   DATA[1995,33] := 0.3065048;
   DATA[1995,34] := 2.0;
   DATA[1995,35] := 250.721;
   DATA[1995,36] := 1.730048;
   DATA[1995,37] := 189.5187;
   DATA[1995,38] := 0.000128152;
   DATA[1995,39] := 1.0;
   DATA[1995,40] := 1.0;
   DATA[1996,0] := 2.641642;
   DATA[1996,1] := 861.0878;
   DATA[1996,2] := 2.0;
   DATA[1996,3] := 2.0;
   DATA[1996,4] := 262.3686;
   DATA[1996,5] := 8.392271;
   DATA[1996,6] := 331.4535;
   DATA[1996,7] := 2.46282;
   DATA[1996,8] := 2.0;
   DATA[1996,9] := 2.0;
   DATA[1996,10] := 2.0;
   DATA[1996,11] := 19.62033;
   DATA[1996,12] := 2.209525;
   DATA[1996,13] := 802.118;
   DATA[1996,14] := 1.0;
   DATA[1996,15] := 2.0;
   DATA[1996,16] := 1.0;
   DATA[1996,17] := 1.0;
   DATA[1996,18] := 1.0;
   DATA[1996,19] := 2.0;
   DATA[1996,20] := 148.808;
   DATA[1996,21] := 154.8834;
   DATA[1996,22] := 1.718387;
   DATA[1996,23] := 827.4033;
   DATA[1996,24] := 2.0;
   DATA[1996,25] := 2.0;
   DATA[1996,26] := 7.874455;
   DATA[1996,27] := 143.9375;
   DATA[1996,28] := 262.0802;
   DATA[1996,29] := 12.07383;
   DATA[1996,30] := 1.728531;
   DATA[1996,31] := 1.303574;
   DATA[1996,32] := 0.7352687;
   DATA[1996,33] := 0.3065048;
   DATA[1996,34] := 2.0;
   DATA[1996,35] := 250.721;
   DATA[1996,36] := 1.730048;
   DATA[1996,37] := 189.5187;
   DATA[1996,38] := 0.000128152;
   DATA[1996,39] := 1.0;
   DATA[1996,40] := 1.0;
   DATA[1997,0] := 2.624988;
   DATA[1997,1] := 861.441;
   DATA[1997,2] := 2.0;
   DATA[1997,3] := 2.0;
   DATA[1997,4] := 262.3686;
   DATA[1997,5] := 8.392271;
   DATA[1997,6] := 331.4535;
   DATA[1997,7] := 2.46423;
   DATA[1997,8] := 2.0;
   DATA[1997,9] := 2.0;
   DATA[1997,10] := 2.0;
   DATA[1997,11] := 19.62033;
   DATA[1997,12] := 2.209525;
   DATA[1997,13] := 802.1982;
   DATA[1997,14] := 1.0;
   DATA[1997,15] := 2.0;
   DATA[1997,16] := 1.0;
   DATA[1997,17] := 1.0;
   DATA[1997,18] := 1.0;
   DATA[1997,19] := 2.0;
   DATA[1997,20] := 148.808;
   DATA[1997,21] := 154.8834;
   DATA[1997,22] := 1.718387;
   DATA[1997,23] := 827.98;
   DATA[1997,24] := 2.0;
   DATA[1997,25] := 2.0;
   DATA[1997,26] := 7.874455;
   DATA[1997,27] := 143.9375;
   DATA[1997,28] := 262.0802;
   DATA[1997,29] := 12.07383;
   DATA[1997,30] := 1.728531;
   DATA[1997,31] := 1.30178;
   DATA[1997,32] := 0.7352687;
   DATA[1997,33] := 0.3065048;
   DATA[1997,34] := 2.0;
   DATA[1997,35] := 250.721;
   DATA[1997,36] := 1.730048;
   DATA[1997,37] := 189.5187;
   DATA[1997,38] := 0.000128152;
   DATA[1997,39] := 1.0;
   DATA[1997,40] := 1.0;
   DATA[1998,0] := 2.617942;
   DATA[1998,1] := 861.4018;
   DATA[1998,2] := 2.0;
   DATA[1998,3] := 2.0;
   DATA[1998,4] := 262.3686;
   DATA[1998,5] := 8.392271;
   DATA[1998,6] := 331.4535;
   DATA[1998,7] := 2.46423;
   DATA[1998,8] := 2.0;
   DATA[1998,9] := 2.0;
   DATA[1998,10] := 2.0;
   DATA[1998,11] := 19.65235;
   DATA[1998,12] := 2.209525;
   DATA[1998,13] := 801.8777;
   DATA[1998,14] := 1.0;
   DATA[1998,15] := 2.0;
   DATA[1998,16] := 1.0;
   DATA[1998,17] := 1.0;
   DATA[1998,18] := 1.0;
   DATA[1998,19] := 2.0;
   DATA[1998,20] := 148.808;
   DATA[1998,21] := 154.8834;
   DATA[1998,22] := 1.719156;
   DATA[1998,23] := 828.2491;
   DATA[1998,24] := 2.0;
   DATA[1998,25] := 2.0;
   DATA[1998,26] := 7.874455;
   DATA[1998,27] := 143.9375;
   DATA[1998,28] := 262.0802;
   DATA[1998,29] := 12.07383;
   DATA[1998,30] := 1.728531;
   DATA[1998,31] := 1.292558;
   DATA[1998,32] := 0.7352687;
   DATA[1998,33] := 0.3065048;
   DATA[1998,34] := 2.0;
   DATA[1998,35] := 250.721;
   DATA[1998,36] := 1.730048;
   DATA[1998,37] := 189.5187;
   DATA[1998,38] := 0.000128152;
   DATA[1998,39] := 1.0;
   DATA[1998,40] := 1.0;
   DATA[1999,0] := 2.611536;
   DATA[1999,1] := 861.0878;
   DATA[1999,2] := 2.0;
   DATA[1999,3] := 2.0;
   DATA[1999,4] := 262.3686;
   DATA[1999,5] := 8.392271;
   DATA[1999,6] := 331.4535;
   DATA[1999,7] := 2.463204;
   DATA[1999,8] := 2.0;
   DATA[1999,9] := 2.0;
   DATA[1999,10] := 2.0;
   DATA[1999,11] := 19.65235;
   DATA[1999,12] := 2.207091;
   DATA[1999,13] := 801.7976;
   DATA[1999,14] := 1.0;
   DATA[1999,15] := 2.0;
   DATA[1999,16] := 1.0;
   DATA[1999,17] := 1.0;
   DATA[1999,18] := 1.0;
   DATA[1999,19] := 2.0;
   DATA[1999,20] := 148.808;
   DATA[1999,21] := 154.8834;
   DATA[1999,22] := 1.720309;
   DATA[1999,23] := 828.5183;
   DATA[1999,24] := 2.0;
   DATA[1999,25] := 2.0;
   DATA[1999,26] := 7.874455;
   DATA[1999,27] := 143.7324;
   DATA[1999,28] := 262.0802;
   DATA[1999,29] := 12.07383;
   DATA[1999,30] := 1.728531;
   DATA[1999,31] := 1.296657;
   DATA[1999,32] := 0.7352687;
   DATA[1999,33] := 0.3065048;
   DATA[1999,34] := 2.0;
   DATA[1999,35] := 250.4807;
   DATA[1999,36] := 1.730048;
   DATA[1999,37] := 189.4867;
   DATA[1999,38] := 0.000128152;
   DATA[1999,39] := 1.0;
   DATA[1999,40] := 1.0;
   DATA[2000,0] := 2.601928;
   DATA[2000,1] := 861.4018;
   DATA[2000,2] := 2.0;
   DATA[2000,3] := 2.0;
   DATA[2000,4] := 262.3686;
   DATA[2000,5] := 8.392271;
   DATA[2000,6] := 331.4535;
   DATA[2000,7] := 2.462564;
   DATA[2000,8] := 2.0;
   DATA[2000,9] := 2.0;
   DATA[2000,10] := 2.0;
   DATA[2000,11] := 19.67476;
   DATA[2000,12] := 2.20645;
   DATA[2000,13] := 801.8777;
   DATA[2000,14] := 1.0;
   DATA[2000,15] := 2.0;
   DATA[2000,16] := 1.0;
   DATA[2000,17] := 1.0;
   DATA[2000,18] := 1.0;
   DATA[2000,19] := 2.0;
   DATA[2000,20] := 148.808;
   DATA[2000,21] := 154.8834;
   DATA[2000,22] := 1.720309;
   DATA[2000,23] := 828.4414;
   DATA[2000,24] := 2.0;
   DATA[2000,25] := 2.0;
   DATA[2000,26] := 7.874455;
   DATA[2000,27] := 143.7324;
   DATA[2000,28] := 262.0802;
   DATA[2000,29] := 12.07383;
   DATA[2000,30] := 1.728531;
   DATA[2000,31] := 1.288075;
   DATA[2000,32] := 0.7352687;
   DATA[2000,33] := 0.3065048;
   DATA[2000,34] := 2.0;
   DATA[2000,35] := 250.4807;
   DATA[2000,36] := 1.730048;
   DATA[2000,37] := 189.4066;
   DATA[2000,38] := 0.000128152;
   DATA[2000,39] := 1.0;
   DATA[2000,40] := 1.0;
   DATA[2001,0] := 2.586555;
   DATA[2001,1] := 861.5195;
   DATA[2001,2] := 2.0;
   DATA[2001,3] := 2.0;
   DATA[2001,4] := 262.3686;
   DATA[2001,5] := 8.392271;
   DATA[2001,6] := 331.4535;
   DATA[2001,7] := 2.46487;
   DATA[2001,8] := 2.0;
   DATA[2001,9] := 2.0;
   DATA[2001,10] := 2.0;
   DATA[2001,11] := 19.73558;
   DATA[2001,12] := 2.205554;
   DATA[2001,13] := 801.4772;
   DATA[2001,14] := 1.0;
   DATA[2001,15] := 2.0;
   DATA[2001,16] := 1.0;
   DATA[2001,17] := 1.0;
   DATA[2001,18] := 1.0;
   DATA[2001,19] := 2.0;
   DATA[2001,20] := 148.808;
   DATA[2001,21] := 154.8834;
   DATA[2001,22] := 1.720309;
   DATA[2001,23] := 828.4799;
   DATA[2001,24] := 2.0;
   DATA[2001,25] := 2.0;
   DATA[2001,26] := 7.874455;
   DATA[2001,27] := 143.7324;
   DATA[2001,28] := 262.0802;
   DATA[2001,29] := 12.07383;
   DATA[2001,30] := 1.728531;
   DATA[2001,31] := 1.282183;
   DATA[2001,32] := 0.7352687;
   DATA[2001,33] := 0.3082983;
   DATA[2001,34] := 2.0;
   DATA[2001,35] := 250.4807;
   DATA[2001,36] := 1.730048;
   DATA[2001,37] := 189.3745;
   DATA[2001,38] := 0.000128152;
   DATA[2001,39] := 1.0;
   DATA[2001,40] := 1.0;
   DATA[2002,0] := 2.570541;
   DATA[2002,1] := 862.0691;
   DATA[2002,2] := 2.0;
   DATA[2002,3] := 2.0;
   DATA[2002,4] := 262.3686;
   DATA[2002,5] := 8.392271;
   DATA[2002,6] := 331.4535;
   DATA[2002,7] := 2.46487;
   DATA[2002,8] := 2.0;
   DATA[2002,9] := 2.0;
   DATA[2002,10] := 2.0;
   DATA[2002,11] := 19.74198;
   DATA[2002,12] := 2.205554;
   DATA[2002,13] := 801.6775;
   DATA[2002,14] := 1.0;
   DATA[2002,15] := 2.0;
   DATA[2002,16] := 1.0;
   DATA[2002,17] := 1.0;
   DATA[2002,18] := 1.0;
   DATA[2002,19] := 2.0;
   DATA[2002,20] := 148.808;
   DATA[2002,21] := 154.8834;
   DATA[2002,22] := 1.720309;
   DATA[2002,23] := 828.4414;
   DATA[2002,24] := 2.0;
   DATA[2002,25] := 2.0;
   DATA[2002,26] := 7.874455;
   DATA[2002,27] := 143.7324;
   DATA[2002,28] := 262.0802;
   DATA[2002,29] := 12.07383;
   DATA[2002,30] := 1.72725;
   DATA[2002,31] := 1.285385;
   DATA[2002,32] := 0.7352687;
   DATA[2002,33] := 0.3082983;
   DATA[2002,34] := 2.0;
   DATA[2002,35] := 250.4807;
   DATA[2002,36] := 1.730048;
   DATA[2002,37] := 189.1823;
   DATA[2002,38] := 0.000128152;
   DATA[2002,39] := 1.0;
   DATA[2002,40] := 1.0;
   DATA[2003,0] := 2.555168;
   DATA[2003,1] := 862.2653;
   DATA[2003,2] := 2.0;
   DATA[2003,3] := 2.0;
   DATA[2003,4] := 262.3686;
   DATA[2003,5] := 8.392271;
   DATA[2003,6] := 331.4535;
   DATA[2003,7] := 2.46487;
   DATA[2003,8] := 2.0;
   DATA[2003,9] := 2.0;
   DATA[2003,10] := 2.0;
   DATA[2003,11] := 19.77079;
   DATA[2003,12] := 2.205554;
   DATA[2003,13] := 801.3571;
   DATA[2003,14] := 1.0;
   DATA[2003,15] := 2.0;
   DATA[2003,16] := 1.0;
   DATA[2003,17] := 1.0;
   DATA[2003,18] := 1.0;
   DATA[2003,19] := 2.0;
   DATA[2003,20] := 148.808;
   DATA[2003,21] := 154.8834;
   DATA[2003,22] := 1.717746;
   DATA[2003,23] := 828.749;
   DATA[2003,24] := 2.0;
   DATA[2003,25] := 2.0;
   DATA[2003,26] := 7.874455;
   DATA[2003,27] := 143.7324;
   DATA[2003,28] := 262.0802;
   DATA[2003,29] := 12.07383;
   DATA[2003,30] := 1.725455;
   DATA[2003,31] := 1.282567;
   DATA[2003,32] := 0.7352687;
   DATA[2003,33] := 0.3082983;
   DATA[2003,34] := 2.0;
   DATA[2003,35] := 250.4005;
   DATA[2003,36] := 1.730048;
   DATA[2003,37] := 189.1823;
   DATA[2003,38] := 0.000128152;
   DATA[2003,39] := 1.0;
   DATA[2003,40] := 1.0;
   DATA[2004,0] := 2.540435;
   DATA[2004,1] := 862.4224;
   DATA[2004,2] := 2.0;
   DATA[2004,3] := 2.0;
   DATA[2004,4] := 262.3686;
   DATA[2004,5] := 8.392271;
   DATA[2004,6] := 331.4535;
   DATA[2004,7] := 2.46487;
   DATA[2004,8] := 2.0;
   DATA[2004,9] := 2.0;
   DATA[2004,10] := 2.0;
   DATA[2004,11] := 19.77079;
   DATA[2004,12] := 2.207347;
   DATA[2004,13] := 801.5573;
   DATA[2004,14] := 1.0;
   DATA[2004,15] := 2.0;
   DATA[2004,16] := 1.0;
   DATA[2004,17] := 1.0;
   DATA[2004,18] := 1.0;
   DATA[2004,19] := 2.0;
   DATA[2004,20] := 148.808;
   DATA[2004,21] := 154.8834;
   DATA[2004,22] := 1.717746;
   DATA[2004,23] := 828.4414;
   DATA[2004,24] := 2.0;
   DATA[2004,25] := 2.0;
   DATA[2004,26] := 7.874455;
   DATA[2004,27] := 143.7324;
   DATA[2004,28] := 262.0802;
   DATA[2004,29] := 12.07383;
   DATA[2004,30] := 1.724814;
   DATA[2004,31] := 1.280389;
   DATA[2004,32] := 0.7352687;
   DATA[2004,33] := 0.3082983;
   DATA[2004,34] := 2.0;
   DATA[2004,35] := 250.4005;
   DATA[2004,36] := 1.730048;
   DATA[2004,37] := 189.1823;
   DATA[2004,38] := 0.000128152;
   DATA[2004,39] := 1.0;
   DATA[2004,40] := 1.0;
   DATA[2005,0] := 2.521859;
   DATA[2005,1] := 862.6186;
   DATA[2005,2] := 2.0;
   DATA[2005,3] := 2.0;
   DATA[2005,4] := 262.3686;
   DATA[2005,5] := 8.392271;
   DATA[2005,6] := 331.4535;
   DATA[2005,7] := 2.463589;
   DATA[2005,8] := 2.0;
   DATA[2005,9] := 2.0;
   DATA[2005,10] := 2.0;
   DATA[2005,11] := 19.77079;
   DATA[2005,12] := 2.207731;
   DATA[2005,13] := 801.9178;
   DATA[2005,14] := 1.0;
   DATA[2005,15] := 2.0;
   DATA[2005,16] := 1.0;
   DATA[2005,17] := 1.0;
   DATA[2005,18] := 1.0;
   DATA[2005,19] := 2.0;
   DATA[2005,20] := 148.808;
   DATA[2005,21] := 154.8834;
   DATA[2005,22] := 1.717105;
   DATA[2005,23] := 828.8259;
   DATA[2005,24] := 2.0;
   DATA[2005,25] := 2.0;
   DATA[2005,26] := 7.874455;
   DATA[2005,27] := 143.8093;
   DATA[2005,28] := 262.0802;
   DATA[2005,29] := 12.07383;
   DATA[2005,30] := 1.724814;
   DATA[2005,31] := 1.273216;
   DATA[2005,32] := 0.7352687;
   DATA[2005,33] := 0.3082983;
   DATA[2005,34] := 2.0;
   DATA[2005,35] := 250.4005;
   DATA[2005,36] := 1.730048;
   DATA[2005,37] := 189.1823;
   DATA[2005,38] := 0.000128152;
   DATA[2005,39] := 1.0;
   DATA[2005,40] := 1.0;
   DATA[2006,0] := 2.507126;
   DATA[2006,1] := 862.3046;
   DATA[2006,2] := 2.0;
   DATA[2006,3] := 2.0;
   DATA[2006,4] := 262.3686;
   DATA[2006,5] := 8.392271;
   DATA[2006,6] := 331.4535;
   DATA[2006,7] := 2.461923;
   DATA[2006,8] := 2.0;
   DATA[2006,9] := 2.0;
   DATA[2006,10] := 2.0;
   DATA[2006,11] := 19.77079;
   DATA[2006,12] := 2.208884;
   DATA[2006,13] := 801.7175;
   DATA[2006,14] := 1.0;
   DATA[2006,15] := 2.0;
   DATA[2006,16] := 1.0;
   DATA[2006,17] := 1.0;
   DATA[2006,18] := 1.0;
   DATA[2006,19] := 2.0;
   DATA[2006,20] := 148.808;
   DATA[2006,21] := 154.8834;
   DATA[2006,22] := 1.71608;
   DATA[2006,23] := 828.7106;
   DATA[2006,24] := 2.0;
   DATA[2006,25] := 2.0;
   DATA[2006,26] := 7.874455;
   DATA[2006,27] := 143.8093;
   DATA[2006,28] := 262.0802;
   DATA[2006,29] := 12.07383;
   DATA[2006,30] := 1.724814;
   DATA[2006,31] := 1.271039;
   DATA[2006,32] := 0.7352687;
   DATA[2006,33] := 0.3082983;
   DATA[2006,34] := 2.0;
   DATA[2006,35] := 250.4005;
   DATA[2006,36] := 1.730048;
   DATA[2006,37] := 189.1823;
   DATA[2006,38] := 0.000128152;
   DATA[2006,39] := 1.0;
   DATA[2006,40] := 1.0;
   DATA[2007,0] := 2.486308;
   DATA[2007,1] := 861.9905;
   DATA[2007,2] := 2.0;
   DATA[2007,3] := 2.0;
   DATA[2007,4] := 262.3686;
   DATA[2007,5] := 8.392271;
   DATA[2007,6] := 331.4535;
   DATA[2007,7] := 2.461539;
   DATA[2007,8] := 2.0;
   DATA[2007,9] := 2.0;
   DATA[2007,10] := 2.0;
   DATA[2007,11] := 19.73238;
   DATA[2007,12] := 2.208884;
   DATA[2007,13] := 801.7976;
   DATA[2007,14] := 1.0;
   DATA[2007,15] := 2.0;
   DATA[2007,16] := 1.0;
   DATA[2007,17] := 1.0;
   DATA[2007,18] := 1.0;
   DATA[2007,19] := 2.0;
   DATA[2007,20] := 148.808;
   DATA[2007,21] := 154.8834;
   DATA[2007,22] := 1.71608;
   DATA[2007,23] := 828.749;
   DATA[2007,24] := 2.0;
   DATA[2007,25] := 2.0;
   DATA[2007,26] := 7.874455;
   DATA[2007,27] := 143.8093;
   DATA[2007,28] := 262.0802;
   DATA[2007,29] := 12.07383;
   DATA[2007,30] := 1.724814;
   DATA[2007,31] := 1.278468;
   DATA[2007,32] := 0.7352687;
   DATA[2007,33] := 0.3082983;
   DATA[2007,34] := 2.0;
   DATA[2007,35] := 250.2563;
   DATA[2007,36] := 1.617916;
   DATA[2007,37] := 189.1823;
   DATA[2007,38] := 0.000128152;
   DATA[2007,39] := 1.0;
   DATA[2007,40] := 1.0;
   DATA[2008,0] := 2.475098;
   DATA[2008,1] := 862.3831;
   DATA[2008,2] := 2.0;
   DATA[2008,3] := 2.0;
   DATA[2008,4] := 262.3686;
   DATA[2008,5] := 8.392271;
   DATA[2008,6] := 331.4535;
   DATA[2008,7] := 2.461539;
   DATA[2008,8] := 2.0;
   DATA[2008,9] := 2.0;
   DATA[2008,10] := 2.0;
   DATA[2008,11] := 19.73238;
   DATA[2008,12] := 2.209013;
   DATA[2008,13] := 801.7976;
   DATA[2008,14] := 1.0;
   DATA[2008,15] := 2.0;
   DATA[2008,16] := 1.0;
   DATA[2008,17] := 1.0;
   DATA[2008,18] := 1.0;
   DATA[2008,19] := 2.0;
   DATA[2008,20] := 148.808;
   DATA[2008,21] := 154.8834;
   DATA[2008,22] := 1.71608;
   DATA[2008,23] := 828.9028;
   DATA[2008,24] := 2.0;
   DATA[2008,25] := 2.0;
   DATA[2008,26] := 7.874455;
   DATA[2008,27] := 143.8093;
   DATA[2008,28] := 262.0802;
   DATA[2008,29] := 12.07383;
   DATA[2008,30] := 1.724814;
   DATA[2008,31] := 1.291789;
   DATA[2008,32] := 0.7352687;
   DATA[2008,33] := 0.3082983;
   DATA[2008,34] := 2.0;
   DATA[2008,35] := 250.2563;
   DATA[2008,36] := 1.617916;
   DATA[2008,37] := 189.1823;
   DATA[2008,38] := 0.000128152;
   DATA[2008,39] := 1.0;
   DATA[2008,40] := 1.0;
   DATA[2009,0] := 2.459405;
   DATA[2009,1] := 862.2653;
   DATA[2009,2] := 2.0;
   DATA[2009,3] := 2.0;
   DATA[2009,4] := 262.3686;
   DATA[2009,5] := 8.392271;
   DATA[2009,6] := 331.4535;
   DATA[2009,7] := 2.46077;
   DATA[2009,8] := 2.0;
   DATA[2009,9] := 2.0;
   DATA[2009,10] := 2.0;
   DATA[2009,11] := 19.72598;
   DATA[2009,12] := 2.210037;
   DATA[2009,13] := 801.4772;
   DATA[2009,14] := 1.0;
   DATA[2009,15] := 2.0;
   DATA[2009,16] := 1.0;
   DATA[2009,17] := 1.0;
   DATA[2009,18] := 1.0;
   DATA[2009,19] := 2.0;
   DATA[2009,20] := 148.808;
   DATA[2009,21] := 154.8834;
   DATA[2009,22] := 1.71608;
   DATA[2009,23] := 829.1335;
   DATA[2009,24] := 2.0;
   DATA[2009,25] := 2.0;
   DATA[2009,26] := 7.874455;
   DATA[2009,27] := 143.8093;
   DATA[2009,28] := 262.0161;
   DATA[2009,29] := 12.07383;
   DATA[2009,30] := 1.724814;
   DATA[2009,31] := 1.301012;
   DATA[2009,32] := 0.7352687;
   DATA[2009,33] := 0.3068891;
   DATA[2009,34] := 2.0;
   DATA[2009,35] := 250.2563;
   DATA[2009,36] := 1.617916;
   DATA[2009,37] := 189.1823;
   DATA[2009,38] := 0.000128152;
   DATA[2009,39] := 1.0;
   DATA[2009,40] := 1.0;
   DATA[2010,0] := 2.436985;
   DATA[2010,1] := 862.4224;
   DATA[2010,2] := 2.0;
   DATA[2010,3] := 2.0;
   DATA[2010,4] := 262.3686;
   DATA[2010,5] := 8.392271;
   DATA[2010,6] := 331.4535;
   DATA[2010,7] := 2.46077;
   DATA[2010,8] := 2.0;
   DATA[2010,9] := 2.0;
   DATA[2010,10] := 2.0;
   DATA[2010,11] := 19.70357;
   DATA[2010,12] := 2.210037;
   DATA[2010,13] := 801.2769;
   DATA[2010,14] := 1.0;
   DATA[2010,15] := 2.0;
   DATA[2010,16] := 1.0;
   DATA[2010,17] := 1.0;
   DATA[2010,18] := 1.0;
   DATA[2010,19] := 2.0;
   DATA[2010,20] := 148.808;
   DATA[2010,21] := 154.8834;
   DATA[2010,22] := 1.71608;
   DATA[2010,23] := 829.2104;
   DATA[2010,24] := 2.0;
   DATA[2010,25] := 2.0;
   DATA[2010,26] := 7.874455;
   DATA[2010,27] := 143.8093;
   DATA[2010,28] := 261.9841;
   DATA[2010,29] := 12.07383;
   DATA[2010,30] := 1.726609;
   DATA[2010,31] := 1.296401;
   DATA[2010,32] := 0.7352687;
   DATA[2010,33] := 0.3068891;
   DATA[2010,34] := 2.0;
   DATA[2010,35] := 250.2563;
   DATA[2010,36] := 1.617916;
   DATA[2010,37] := 189.1823;
   DATA[2010,38] := 0.000128152;
   DATA[2010,39] := 1.0;
   DATA[2010,40] := 1.0;
   DATA[2011,0] := 2.424174;
   DATA[2011,1] := 862.1868;
   DATA[2011,2] := 2.0;
   DATA[2011,3] := 2.0;
   DATA[2011,4] := 262.3686;
   DATA[2011,5] := 8.392271;
   DATA[2011,6] := 331.4535;
   DATA[2011,7] := 2.46077;
   DATA[2011,8] := 2.0;
   DATA[2011,9] := 2.0;
   DATA[2011,10] := 2.0;
   DATA[2011,11] := 19.70357;
   DATA[2011,12] := 2.210037;
   DATA[2011,13] := 801.2769;
   DATA[2011,14] := 1.0;
   DATA[2011,15] := 2.0;
   DATA[2011,16] := 1.0;
   DATA[2011,17] := 1.0;
   DATA[2011,18] := 1.0;
   DATA[2011,19] := 2.0;
   DATA[2011,20] := 148.808;
   DATA[2011,21] := 154.8065;
   DATA[2011,22] := 1.717746;
   DATA[2011,23] := 829.595;
   DATA[2011,24] := 2.0;
   DATA[2011,25] := 2.0;
   DATA[2011,26] := 7.874455;
   DATA[2011,27] := 143.8093;
   DATA[2011,28] := 261.9841;
   DATA[2011,29] := 12.07383;
   DATA[2011,30] := 1.729428;
   DATA[2011,31] := 1.298962;
   DATA[2011,32] := 0.7352687;
   DATA[2011,33] := 0.3068891;
   DATA[2011,34] := 2.0;
   DATA[2011,35] := 250.2563;
   DATA[2011,36] := 1.69801;
   DATA[2011,37] := 189.1823;
   DATA[2011,38] := 0.000128152;
   DATA[2011,39] := 1.0;
   DATA[2011,40] := 1.0;
   DATA[2012,0] := 2.41937;
   DATA[2012,1] := 862.3046;
   DATA[2012,2] := 2.0;
   DATA[2012,3] := 2.0;
   DATA[2012,4] := 262.3686;
   DATA[2012,5] := 8.392271;
   DATA[2012,6] := 331.4535;
   DATA[2012,7] := 2.46077;
   DATA[2012,8] := 2.0;
   DATA[2012,9] := 2.0;
   DATA[2012,10] := 2.0;
   DATA[2012,11] := 19.76759;
   DATA[2012,12] := 2.210037;
   DATA[2012,13] := 801.1167;
   DATA[2012,14] := 1.0;
   DATA[2012,15] := 2.0;
   DATA[2012,16] := 1.0;
   DATA[2012,17] := 1.0;
   DATA[2012,18] := 1.0;
   DATA[2012,19] := 2.0;
   DATA[2012,20] := 148.808;
   DATA[2012,21] := 154.7552;
   DATA[2012,22] := 1.717746;
   DATA[2012,23] := 829.6719;
   DATA[2012,24] := 2.0;
   DATA[2012,25] := 2.0;
   DATA[2012,26] := 7.874455;
   DATA[2012,27] := 143.8093;
   DATA[2012,28] := 261.9841;
   DATA[2012,29] := 12.07383;
   DATA[2012,30] := 1.729428;
   DATA[2012,31] := 1.293967;
   DATA[2012,32] := 0.7352687;
   DATA[2012,33] := 0.3065048;
   DATA[2012,34] := 2.0;
   DATA[2012,35] := 250.2563;
   DATA[2012,36] := 1.69801;
   DATA[2012,37] := 189.1823;
   DATA[2012,38] := 0.000128152;
   DATA[2012,39] := 1.0;
   DATA[2012,40] := 1.0;
   DATA[2013,0] := 2.41937;
   DATA[2013,1] := 862.2653;
   DATA[2013,2] := 2.0;
   DATA[2013,3] := 2.0;
   DATA[2013,4] := 262.3686;
   DATA[2013,5] := 8.392271;
   DATA[2013,6] := 331.4535;
   DATA[2013,7] := 2.463461;
   DATA[2013,8] := 2.0;
   DATA[2013,9] := 2.0;
   DATA[2013,10] := 2.0;
   DATA[2013,11] := 19.77079;
   DATA[2013,12] := 2.210037;
   DATA[2013,13] := 800.7963;
   DATA[2013,14] := 1.0;
   DATA[2013,15] := 2.0;
   DATA[2013,16] := 1.0;
   DATA[2013,17] := 1.0;
   DATA[2013,18] := 1.0;
   DATA[2013,19] := 2.0;
   DATA[2013,20] := 148.808;
   DATA[2013,21] := 154.7552;
   DATA[2013,22] := 1.717746;
   DATA[2013,23] := 829.8257;
   DATA[2013,24] := 2.0;
   DATA[2013,25] := 2.0;
   DATA[2013,26] := 7.874455;
   DATA[2013,27] := 143.8093;
   DATA[2013,28] := 261.9841;
   DATA[2013,29] := 12.07383;
   DATA[2013,30] := 1.729428;
   DATA[2013,31] := 1.29243;
   DATA[2013,32] := 0.7352687;
   DATA[2013,33] := 0.3065048;
   DATA[2013,34] := 2.0;
   DATA[2013,35] := 250.4166;
   DATA[2013,36] := 1.69801;
   DATA[2013,37] := 189.1823;
   DATA[2013,38] := 0.000128152;
   DATA[2013,39] := 1.0;
   DATA[2013,40] := 1.0;
   DATA[2014,0] := 2.452679;
   DATA[2014,1] := 862.5793;
   DATA[2014,2] := 2.0;
   DATA[2014,3] := 2.0;
   DATA[2014,4] := 262.3686;
   DATA[2014,5] := 8.392271;
   DATA[2014,6] := 331.4535;
   DATA[2014,7] := 2.463461;
   DATA[2014,8] := 2.0;
   DATA[2014,9] := 2.0;
   DATA[2014,10] := 2.0;
   DATA[2014,11] := 19.77079;
   DATA[2014,12] := 2.208884;
   DATA[2014,13] := 800.7162;
   DATA[2014,14] := 1.0;
   DATA[2014,15] := 2.0;
   DATA[2014,16] := 1.0;
   DATA[2014,17] := 1.0;
   DATA[2014,18] := 1.0;
   DATA[2014,19] := 2.0;
   DATA[2014,20] := 148.808;
   DATA[2014,21] := 154.7552;
   DATA[2014,22] := 1.717746;
   DATA[2014,23] := 829.9795;
   DATA[2014,24] := 2.0;
   DATA[2014,25] := 2.0;
   DATA[2014,26] := 7.874455;
   DATA[2014,27] := 143.8093;
   DATA[2014,28] := 261.9841;
   DATA[2014,29] := 12.07383;
   DATA[2014,30] := 1.729428;
   DATA[2014,31] := 1.297554;
   DATA[2014,32] := 0.7352687;
   DATA[2014,33] := 0.3065048;
   DATA[2014,34] := 2.0;
   DATA[2014,35] := 250.4166;
   DATA[2014,36] := 1.69801;
   DATA[2014,37] := 189.1823;
   DATA[2014,38] := 0.000128152;
   DATA[2014,39] := 1.0;
   DATA[2014,40] := 1.0;
   DATA[2015,0] := 2.494635;
   DATA[2015,1] := 862.2261;
   DATA[2015,2] := 2.0;
   DATA[2015,3] := 2.0;
   DATA[2015,4] := 262.3686;
   DATA[2015,5] := 8.392271;
   DATA[2015,6] := 331.4535;
   DATA[2015,7] := 2.463461;
   DATA[2015,8] := 2.0;
   DATA[2015,9] := 2.0;
   DATA[2015,10] := 2.0;
   DATA[2015,11] := 19.77079;
   DATA[2015,12] := 2.208884;
   DATA[2015,13] := 800.596;
   DATA[2015,14] := 1.0;
   DATA[2015,15] := 2.0;
   DATA[2015,16] := 1.0;
   DATA[2015,17] := 1.0;
   DATA[2015,18] := 1.0;
   DATA[2015,19] := 2.0;
   DATA[2015,20] := 148.808;
   DATA[2015,21] := 154.7552;
   DATA[2015,22] := 1.719156;
   DATA[2015,23] := 830.0564;
   DATA[2015,24] := 2.0;
   DATA[2015,25] := 2.0;
   DATA[2015,26] := 7.874455;
   DATA[2015,27] := 143.8093;
   DATA[2015,28] := 261.9841;
   DATA[2015,29] := 12.07383;
   DATA[2015,30] := 1.729428;
   DATA[2015,31] := 1.296273;
   DATA[2015,32] := 0.7352687;
   DATA[2015,33] := 0.3065048;
   DATA[2015,34] := 2.0;
   DATA[2015,35] := 250.4166;
   DATA[2015,36] := 1.69801;
   DATA[2015,37] := 189.1823;
   DATA[2015,38] := 0.000128152;
   DATA[2015,39] := 1.0;
   DATA[2015,40] := 1.0;
   DATA[2016,0] := 2.537232;
   DATA[2016,1] := 862.5793;
   DATA[2016,2] := 2.0;
   DATA[2016,3] := 2.0;
   DATA[2016,4] := 262.3686;
   DATA[2016,5] := 8.392271;
   DATA[2016,6] := 331.4535;
   DATA[2016,7] := 2.463461;
   DATA[2016,8] := 2.0;
   DATA[2016,9] := 2.0;
   DATA[2016,10] := 2.0;
   DATA[2016,11] := 19.77079;
   DATA[2016,12] := 2.210166;
   DATA[2016,13] := 800.7162;
   DATA[2016,14] := 1.0;
   DATA[2016,15] := 2.0;
   DATA[2016,16] := 1.0;
   DATA[2016,17] := 1.0;
   DATA[2016,18] := 1.0;
   DATA[2016,19] := 2.0;
   DATA[2016,20] := 148.808;
   DATA[2016,21] := 154.7552;
   DATA[2016,22] := 1.719156;
   DATA[2016,23] := 830.2871;
   DATA[2016,24] := 2.0;
   DATA[2016,25] := 2.0;
   DATA[2016,26] := 7.874455;
   DATA[2016,27] := 143.8093;
   DATA[2016,28] := 261.9841;
   DATA[2016,29] := 12.07383;
   DATA[2016,30] := 1.729428;
   DATA[2016,31] := 1.3005;
   DATA[2016,32] := 0.7352687;
   DATA[2016,33] := 0.3065048;
   DATA[2016,34] := 2.0;
   DATA[2016,35] := 250.4166;
   DATA[2016,36] := 1.69801;
   DATA[2016,37] := 189.1823;
   DATA[2016,38] := 0.000128152;
   DATA[2016,39] := 1.0;
   DATA[2016,40] := 1.0;
   DATA[2017,0] := 2.572142;
   DATA[2017,1] := 862.1868;
   DATA[2017,2] := 2.0;
   DATA[2017,3] := 2.0;
   DATA[2017,4] := 262.3686;
   DATA[2017,5] := 8.392271;
   DATA[2017,6] := 331.4535;
   DATA[2017,7] := 2.463461;
   DATA[2017,8] := 2.0;
   DATA[2017,9] := 2.0;
   DATA[2017,10] := 2.0;
   DATA[2017,11] := 19.7996;
   DATA[2017,12] := 2.210678;
   DATA[2017,13] := 800.596;
   DATA[2017,14] := 1.0;
   DATA[2017,15] := 2.0;
   DATA[2017,16] := 1.0;
   DATA[2017,17] := 1.0;
   DATA[2017,18] := 1.0;
   DATA[2017,19] := 2.0;
   DATA[2017,20] := 148.808;
   DATA[2017,21] := 154.7552;
   DATA[2017,22] := 1.719156;
   DATA[2017,23] := 830.4025;
   DATA[2017,24] := 2.0;
   DATA[2017,25] := 2.0;
   DATA[2017,26] := 7.874455;
   DATA[2017,27] := 143.8093;
   DATA[2017,28] := 261.9841;
   DATA[2017,29] := 12.07383;
   DATA[2017,30] := 1.729428;
   DATA[2017,31] := 1.30178;
   DATA[2017,32] := 0.7352687;
   DATA[2017,33] := 0.3065048;
   DATA[2017,34] := 2.0;
   DATA[2017,35] := 250.3365;
   DATA[2017,36] := 1.69801;
   DATA[2017,37] := 189.1823;
   DATA[2017,38] := 0.000128152;
   DATA[2017,39] := 1.0;
   DATA[2017,40] := 1.0;
   DATA[2018,0] := 2.607373;
   DATA[2018,1] := 862.3831;
   DATA[2018,2] := 2.0;
   DATA[2018,3] := 2.0;
   DATA[2018,4] := 262.3686;
   DATA[2018,5] := 8.392271;
   DATA[2018,6] := 331.4535;
   DATA[2018,7] := 2.463461;
   DATA[2018,8] := 2.0;
   DATA[2018,9] := 2.0;
   DATA[2018,10] := 2.0;
   DATA[2018,11] := 19.81561;
   DATA[2018,12] := 2.210678;
   DATA[2018,13] := 799.9952;
   DATA[2018,14] := 1.0;
   DATA[2018,15] := 2.0;
   DATA[2018,16] := 1.0;
   DATA[2018,17] := 1.0;
   DATA[2018,18] := 1.0;
   DATA[2018,19] := 2.0;
   DATA[2018,20] := 148.808;
   DATA[2018,21] := 154.7552;
   DATA[2018,22] := 1.719156;
   DATA[2018,23] := 830.5947;
   DATA[2018,24] := 2.0;
   DATA[2018,25] := 2.0;
   DATA[2018,26] := 7.874455;
   DATA[2018,27] := 143.8093;
   DATA[2018,28] := 261.9841;
   DATA[2018,29] := 12.07383;
   DATA[2018,30] := 1.729428;
   DATA[2018,31] := 1.293839;
   DATA[2018,32] := 0.7352687;
   DATA[2018,33] := 0.3065048;
   DATA[2018,34] := 2.0;
   DATA[2018,35] := 250.3365;
   DATA[2018,36] := 1.69801;
   DATA[2018,37] := 189.1823;
   DATA[2018,38] := 0.000128152;
   DATA[2018,39] := 1.0;
   DATA[2018,40] := 1.0;
   DATA[2019,0] := 2.630753;
   DATA[2019,1] := 862.5009;
   DATA[2019,2] := 2.0;
   DATA[2019,3] := 2.0;
   DATA[2019,4] := 262.3686;
   DATA[2019,5] := 8.392271;
   DATA[2019,6] := 331.3509;
   DATA[2019,7] := 2.463461;
   DATA[2019,8] := 2.0;
   DATA[2019,9] := 2.0;
   DATA[2019,10] := 2.0;
   DATA[2019,11] := 19.81561;
   DATA[2019,12] := 2.210678;
   DATA[2019,13] := 800.4758;
   DATA[2019,14] := 1.0;
   DATA[2019,15] := 2.0;
   DATA[2019,16] := 1.0;
   DATA[2019,17] := 1.0;
   DATA[2019,18] := 1.0;
   DATA[2019,19] := 2.0;
   DATA[2019,20] := 148.808;
   DATA[2019,21] := 154.7552;
   DATA[2019,22] := 1.719156;
   DATA[2019,23] := 830.7485;
   DATA[2019,24] := 2.0;
   DATA[2019,25] := 2.0;
   DATA[2019,26] := 7.874455;
   DATA[2019,27] := 143.8093;
   DATA[2019,28] := 261.9841;
   DATA[2019,29] := 12.07383;
   DATA[2019,30] := 1.729428;
   DATA[2019,31] := 1.291789;
   DATA[2019,32] := 0.7352687;
   DATA[2019,33] := 0.3081062;
   DATA[2019,34] := 2.0;
   DATA[2019,35] := 250.3365;
   DATA[2019,36] := 1.69801;
   DATA[2019,37] := 189.1823;
   DATA[2019,38] := 0.000128152;
   DATA[2019,39] := 1.0;
   DATA[2019,40] := 1.0;
   DATA[2020,0] := 2.653172;
   DATA[2020,1] := 862.2261;
   DATA[2020,2] := 2.0;
   DATA[2020,3] := 2.0;
   DATA[2020,4] := 262.3686;
   DATA[2020,5] := 8.392271;
   DATA[2020,6] := 331.3509;
   DATA[2020,7] := 2.463461;
   DATA[2020,8] := 2.0;
   DATA[2020,9] := 2.0;
   DATA[2020,10] := 2.0;
   DATA[2020,11] := 19.81561;
   DATA[2020,12] := 2.208884;
   DATA[2020,13] := 800.1955;
   DATA[2020,14] := 1.0;
   DATA[2020,15] := 2.0;
   DATA[2020,16] := 1.0;
   DATA[2020,17] := 1.0;
   DATA[2020,18] := 1.0;
   DATA[2020,19] := 2.0;
   DATA[2020,20] := 148.808;
   DATA[2020,21] := 154.7552;
   DATA[2020,22] := 1.719156;
   DATA[2020,23] := 830.9408;
   DATA[2020,24] := 2.0;
   DATA[2020,25] := 2.0;
   DATA[2020,26] := 7.874455;
   DATA[2020,27] := 143.8093;
   DATA[2020,28] := 261.9841;
   DATA[2020,29] := 12.07383;
   DATA[2020,30] := 1.728147;
   DATA[2020,31] := 1.291789;
   DATA[2020,32] := 0.7352687;
   DATA[2020,33] := 0.3084905;
   DATA[2020,34] := 2.0;
   DATA[2020,35] := 250.3365;
   DATA[2020,36] := 1.69801;
   DATA[2020,37] := 189.1823;
   DATA[2020,38] := 0.000128152;
   DATA[2020,39] := 1.0;
   DATA[2020,40] := 1.0;
   DATA[2021,0] := 2.654133;
   DATA[2021,1] := 862.4224;
   DATA[2021,2] := 2.0;
   DATA[2021,3] := 2.0;
   DATA[2021,4] := 262.3686;
   DATA[2021,5] := 8.392271;
   DATA[2021,6] := 331.3509;
   DATA[2021,7] := 2.462179;
   DATA[2021,8] := 2.0;
   DATA[2021,9] := 2.0;
   DATA[2021,10] := 2.0;
   DATA[2021,11] := 19.81561;
   DATA[2021,12] := 2.208884;
   DATA[2021,13] := 800.2756;
   DATA[2021,14] := 1.0;
   DATA[2021,15] := 2.0;
   DATA[2021,16] := 1.0;
   DATA[2021,17] := 1.0;
   DATA[2021,18] := 1.0;
   DATA[2021,19] := 2.0;
   DATA[2021,20] := 148.808;
   DATA[2021,21] := 154.7552;
   DATA[2021,22] := 1.717361;
   DATA[2021,23] := 830.9408;
   DATA[2021,24] := 2.0;
   DATA[2021,25] := 2.0;
   DATA[2021,26] := 7.874455;
   DATA[2021,27] := 143.8093;
   DATA[2021,28] := 261.9841;
   DATA[2021,29] := 12.07383;
   DATA[2021,30] := 1.728147;
   DATA[2021,31] := 1.282951;
   DATA[2021,32] := 0.7352687;
   DATA[2021,33] := 0.3084905;
   DATA[2021,34] := 2.0;
   DATA[2021,35] := 250.3044;
   DATA[2021,36] := 1.69801;
   DATA[2021,37] := 189.1823;
   DATA[2021,38] := 0.000128152;
   DATA[2021,39] := 1.0;
   DATA[2021,40] := 1.0;
   DATA[2022,0] := 2.645806;
   DATA[2022,1] := 862.0298;
   DATA[2022,2] := 2.0;
   DATA[2022,3] := 2.0;
   DATA[2022,4] := 262.3686;
   DATA[2022,5] := 8.392271;
   DATA[2022,6] := 331.3509;
   DATA[2022,7] := 2.462179;
   DATA[2022,8] := 2.0;
   DATA[2022,9] := 2.0;
   DATA[2022,10] := 2.0;
   DATA[2022,11] := 19.81561;
   DATA[2022,12] := 2.208884;
   DATA[2022,13] := 800.3958;
   DATA[2022,14] := 1.0;
   DATA[2022,15] := 2.0;
   DATA[2022,16] := 1.0;
   DATA[2022,17] := 1.0;
   DATA[2022,18] := 1.0;
   DATA[2022,19] := 2.0;
   DATA[2022,20] := 148.808;
   DATA[2022,21] := 154.6526;
   DATA[2022,22] := 1.717361;
   DATA[2022,23] := 831.0177;
   DATA[2022,24] := 2.0;
   DATA[2022,25] := 2.0;
   DATA[2022,26] := 7.874455;
   DATA[2022,27] := 143.8093;
   DATA[2022,28] := 261.9841;
   DATA[2022,29] := 12.07383;
   DATA[2022,30] := 1.726737;
   DATA[2022,31] := 1.287562;
   DATA[2022,32] := 0.7352687;
   DATA[2022,33] := 0.3084905;
   DATA[2022,34] := 2.0;
   DATA[2022,35] := 250.2243;
   DATA[2022,36] := 1.69801;
   DATA[2022,37] := 189.1823;
   DATA[2022,38] := 0.000128152;
   DATA[2022,39] := 1.0;
   DATA[2022,40] := 1.0;
   DATA[2023,0] := 2.623707;
   DATA[2023,1] := 862.3046;
   DATA[2023,2] := 2.0;
   DATA[2023,3] := 2.0;
   DATA[2023,4] := 262.3686;
   DATA[2023,5] := 8.392271;
   DATA[2023,6] := 331.3509;
   DATA[2023,7] := 2.462179;
   DATA[2023,8] := 2.0;
   DATA[2023,9] := 2.0;
   DATA[2023,10] := 2.0;
   DATA[2023,11] := 19.81561;
   DATA[2023,12] := 2.208884;
   DATA[2023,13] := 800.3958;
   DATA[2023,14] := 1.0;
   DATA[2023,15] := 2.0;
   DATA[2023,16] := 1.0;
   DATA[2023,17] := 1.0;
   DATA[2023,18] := 1.0;
   DATA[2023,19] := 2.0;
   DATA[2023,20] := 148.808;
   DATA[2023,21] := 154.6526;
   DATA[2023,22] := 1.717361;
   DATA[2023,23] := 830.6332;
   DATA[2023,24] := 2.0;
   DATA[2023,25] := 2.0;
   DATA[2023,26] := 7.874455;
   DATA[2023,27] := 143.8093;
   DATA[2023,28] := 262.1764;
   DATA[2023,29] := 12.07383;
   DATA[2023,30] := 1.726224;
   DATA[2023,31] := 1.277956;
   DATA[2023,32] := 0.7352687;
   DATA[2023,33] := 0.3084905;
   DATA[2023,34] := 2.0;
   DATA[2023,35] := 250.2243;
   DATA[2023,36] := 1.69801;
   DATA[2023,37] := 189.1823;
   DATA[2023,38] := 0.000128152;
   DATA[2023,39] := 1.0;
   DATA[2023,40] := 1.0;
   DATA[2024,0] := 2.612818;
   DATA[2024,1] := 862.1083;
   DATA[2024,2] := 2.0;
   DATA[2024,3] := 2.0;
   DATA[2024,4] := 262.3686;
   DATA[2024,5] := 8.392271;
   DATA[2024,6] := 331.3509;
   DATA[2024,7] := 2.462179;
   DATA[2024,8] := 2.0;
   DATA[2024,9] := 2.0;
   DATA[2024,10] := 2.0;
   DATA[2024,11] := 19.87003;
   DATA[2024,12] := 2.208884;
   DATA[2024,13] := 800.3958;
   DATA[2024,14] := 1.0;
   DATA[2024,15] := 2.0;
   DATA[2024,16] := 1.0;
   DATA[2024,17] := 1.0;
   DATA[2024,18] := 1.0;
   DATA[2024,19] := 2.0;
   DATA[2024,20] := 148.808;
   DATA[2024,21] := 154.6526;
   DATA[2024,22] := 1.717361;
   DATA[2024,23] := 831.1331;
   DATA[2024,24] := 2.0;
   DATA[2024,25] := 2.0;
   DATA[2024,26] := 7.874455;
   DATA[2024,27] := 143.8093;
   DATA[2024,28] := 262.1764;
   DATA[2024,29] := 12.07383;
   DATA[2024,30] := 1.726224;
   DATA[2024,31] := 1.271935;
   DATA[2024,32] := 0.7352687;
   DATA[2024,33] := 0.3084905;
   DATA[2024,34] := 2.0;
   DATA[2024,35] := 250.2243;
   DATA[2024,36] := 1.69801;
   DATA[2024,37] := 189.1823;
   DATA[2024,38] := 0.000128152;
   DATA[2024,39] := 1.0;
   DATA[2024,40] := 1.0;
   DATA[2025,0] := 2.612818;
   DATA[2025,1] := 862.5009;
   DATA[2025,2] := 2.0;
   DATA[2025,3] := 2.0;
   DATA[2025,4] := 262.3686;
   DATA[2025,5] := 8.392271;
   DATA[2025,6] := 331.3509;
   DATA[2025,7] := 2.462179;
   DATA[2025,8] := 2.0;
   DATA[2025,9] := 2.0;
   DATA[2025,10] := 2.0;
   DATA[2025,11] := 19.91165;
   DATA[2025,12] := 2.208884;
   DATA[2025,13] := 800.9164;
   DATA[2025,14] := 1.0;
   DATA[2025,15] := 2.0;
   DATA[2025,16] := 1.0;
   DATA[2025,17] := 1.0;
   DATA[2025,18] := 1.0;
   DATA[2025,19] := 2.0;
   DATA[2025,20] := 148.808;
   DATA[2025,21] := 154.6526;
   DATA[2025,22] := 1.717361;
   DATA[2025,23] := 831.0177;
   DATA[2025,24] := 2.0;
   DATA[2025,25] := 2.0;
   DATA[2025,26] := 7.874455;
   DATA[2025,27] := 143.8093;
   DATA[2025,28] := 262.1764;
   DATA[2025,29] := 12.07383;
   DATA[2025,30] := 1.726224;
   DATA[2025,31] := 1.280517;
   DATA[2025,32] := 0.7352687;
   DATA[2025,33] := 0.3084905;
   DATA[2025,34] := 2.0;
   DATA[2025,35] := 250.2243;
   DATA[2025,36] := 1.69801;
   DATA[2025,37] := 189.1823;
   DATA[2025,38] := 0.000128152;
   DATA[2025,39] := 1.0;
   DATA[2025,40] := 1.0;
   DATA[2026,0] := 2.600967;
   DATA[2026,1] := 862.3831;
   DATA[2026,2] := 2.0;
   DATA[2026,3] := 2.0;
   DATA[2026,4] := 262.3686;
   DATA[2026,5] := 8.392271;
   DATA[2026,6] := 331.1971;
   DATA[2026,7] := 2.462179;
   DATA[2026,8] := 2.0;
   DATA[2026,9] := 2.0;
   DATA[2026,10] := 2.0;
   DATA[2026,11] := 19.92445;
   DATA[2026,12] := 2.208884;
   DATA[2026,13] := 800.7562;
   DATA[2026,14] := 1.0;
   DATA[2026,15] := 2.0;
   DATA[2026,16] := 1.0;
   DATA[2026,17] := 1.0;
   DATA[2026,18] := 1.0;
   DATA[2026,19] := 2.0;
   DATA[2026,20] := 148.808;
   DATA[2026,21] := 154.6526;
   DATA[2026,22] := 1.717361;
   DATA[2026,23] := 830.9792;
   DATA[2026,24] := 2.0;
   DATA[2026,25] := 2.0;
   DATA[2026,26] := 7.874455;
   DATA[2026,27] := 143.8093;
   DATA[2026,28] := 262.1764;
   DATA[2026,29] := 12.07383;
   DATA[2026,30] := 1.727378;
   DATA[2026,31] := 1.286922;
   DATA[2026,32] := 0.7374452;
   DATA[2026,33] := 0.3084905;
   DATA[2026,34] := 2.0;
   DATA[2026,35] := 250.2243;
   DATA[2026,36] := 1.69801;
   DATA[2026,37] := 189.1823;
   DATA[2026,38] := 0.000128152;
   DATA[2026,39] := 1.0;
   DATA[2026,40] := 1.0;
   DATA[2027,0] := 2.585274;
   DATA[2027,1] := 862.6971;
   DATA[2027,2] := 2.0;
   DATA[2027,3] := 2.0;
   DATA[2027,4] := 262.3686;
   DATA[2027,5] := 8.392271;
   DATA[2027,6] := 331.1971;
   DATA[2027,7] := 2.462179;
   DATA[2027,8] := 2.0;
   DATA[2027,9] := 2.0;
   DATA[2027,10] := 2.0;
   DATA[2027,11] := 19.92445;
   DATA[2027,12] := 2.208884;
   DATA[2027,13] := 801.1167;
   DATA[2027,14] := 1.0;
   DATA[2027,15] := 2.0;
   DATA[2027,16] := 1.0;
   DATA[2027,17] := 1.0;
   DATA[2027,18] := 1.0;
   DATA[2027,19] := 2.0;
   DATA[2027,20] := 148.808;
   DATA[2027,21] := 154.6526;
   DATA[2027,22] := 1.717361;
   DATA[2027,23] := 831.5176;
   DATA[2027,24] := 2.0;
   DATA[2027,25] := 2.0;
   DATA[2027,26] := 7.874455;
   DATA[2027,27] := 143.8093;
   DATA[2027,28] := 262.1764;
   DATA[2027,29] := 12.07383;
   DATA[2027,30] := 1.727378;
   DATA[2027,31] := 1.301652;
   DATA[2027,32] := 0.7374452;
   DATA[2027,33] := 0.3084905;
   DATA[2027,34] := 2.0;
   DATA[2027,35] := 250.2243;
   DATA[2027,36] := 1.69801;
   DATA[2027,37] := 189.1823;
   DATA[2027,38] := 0.000128152;
   DATA[2027,39] := 1.0;
   DATA[2027,40] := 1.0;
   DATA[2028,0] := 2.567979;
   DATA[2028,1] := 862.4224;
   DATA[2028,2] := 2.0;
   DATA[2028,3] := 2.0;
   DATA[2028,4] := 262.3686;
   DATA[2028,5] := 8.392271;
   DATA[2028,6] := 331.1971;
   DATA[2028,7] := 2.462179;
   DATA[2028,8] := 2.0;
   DATA[2028,9] := 2.0;
   DATA[2028,10] := 2.0;
   DATA[2028,11] := 19.89244;
   DATA[2028,12] := 2.208884;
   DATA[2028,13] := 801.4772;
   DATA[2028,14] := 1.0;
   DATA[2028,15] := 2.0;
   DATA[2028,16] := 1.0;
   DATA[2028,17] := 1.0;
   DATA[2028,18] := 1.0;
   DATA[2028,19] := 2.0;
   DATA[2028,20] := 148.808;
   DATA[2028,21] := 154.6526;
   DATA[2028,22] := 1.717361;
   DATA[2028,23] := 831.1331;
   DATA[2028,24] := 2.0;
   DATA[2028,25] := 2.0;
   DATA[2028,26] := 7.874455;
   DATA[2028,27] := 143.8093;
   DATA[2028,28] := 262.1764;
   DATA[2028,29] := 12.07383;
   DATA[2028,30] := 1.727378;
   DATA[2028,31] := 1.302421;
   DATA[2028,32] := 0.7374452;
   DATA[2028,33] := 0.3084905;
   DATA[2028,34] := 2.0;
   DATA[2028,35] := 250.2243;
   DATA[2028,36] := 1.69801;
   DATA[2028,37] := 189.1823;
   DATA[2028,38] := 0.000128152;
   DATA[2028,39] := 1.0;
   DATA[2028,40] := 1.0;
   DATA[2029,0] := 2.557089;
   DATA[2029,1] := 862.4616;
   DATA[2029,2] := 2.0;
   DATA[2029,3] := 2.0;
   DATA[2029,4] := 262.3686;
   DATA[2029,5] := 8.393232;
   DATA[2029,6] := 331.1971;
   DATA[2029,7] := 2.462179;
   DATA[2029,8] := 2.0;
   DATA[2029,9] := 2.0;
   DATA[2029,10] := 2.0;
   DATA[2029,11] := 19.84762;
   DATA[2029,12] := 2.208884;
   DATA[2029,13] := 801.317;
   DATA[2029,14] := 1.0;
   DATA[2029,15] := 2.0;
   DATA[2029,16] := 1.0;
   DATA[2029,17] := 1.0;
   DATA[2029,18] := 1.0;
   DATA[2029,19] := 2.0;
   DATA[2029,20] := 148.808;
   DATA[2029,21] := 154.909;
   DATA[2029,22] := 1.717361;
   DATA[2029,23] := 831.1331;
   DATA[2029,24] := 2.0;
   DATA[2029,25] := 2.0;
   DATA[2029,26] := 7.874455;
   DATA[2029,27] := 143.8093;
   DATA[2029,28] := 262.1764;
   DATA[2029,29] := 12.07383;
   DATA[2029,30] := 1.727378;
   DATA[2029,31] := 1.291405;
   DATA[2029,32] := 0.7374452;
   DATA[2029,33] := 0.3084905;
   DATA[2029,34] := 2.0;
   DATA[2029,35] := 250.2243;
   DATA[2029,36] := 1.69801;
   DATA[2029,37] := 189.1823;
   DATA[2029,38] := 0.000128152;
   DATA[2029,39] := 1.0;
   DATA[2029,40] := 1.0;
   DATA[2030,0] := 2.540755;
   DATA[2030,1] := 862.3831;
   DATA[2030,2] := 2.0;
   DATA[2030,3] := 2.0;
   DATA[2030,4] := 262.3686;
   DATA[2030,5] := 8.395155;
   DATA[2030,6] := 331.1971;
   DATA[2030,7] := 2.462179;
   DATA[2030,8] := 2.0;
   DATA[2030,9] := 2.0;
   DATA[2030,10] := 2.0;
   DATA[2030,11] := 19.7996;
   DATA[2030,12] := 2.209653;
   DATA[2030,13] := 801.6775;
   DATA[2030,14] := 1.0;
   DATA[2030,15] := 2.0;
   DATA[2030,16] := 1.0;
   DATA[2030,17] := 1.0;
   DATA[2030,18] := 1.0;
   DATA[2030,19] := 2.0;
   DATA[2030,20] := 148.808;
   DATA[2030,21] := 154.909;
   DATA[2030,22] := 1.718643;
   DATA[2030,23] := 831.2484;
   DATA[2030,24] := 2.0;
   DATA[2030,25] := 2.0;
   DATA[2030,26] := 7.874455;
   DATA[2030,27] := 143.8093;
   DATA[2030,28] := 262.1764;
   DATA[2030,29] := 12.07383;
   DATA[2030,30] := 1.726609;
   DATA[2030,31] := 1.291277;
   DATA[2030,32] := 0.7355248;
   DATA[2030,33] := 0.3084905;
   DATA[2030,34] := 2.0;
   DATA[2030,35] := 250.2243;
   DATA[2030,36] := 1.69801;
   DATA[2030,37] := 189.1823;
   DATA[2030,38] := 0.000128152;
   DATA[2030,39] := 1.0;
   DATA[2030,40] := 1.0;
   DATA[2031,0] := 2.52314;
   DATA[2031,1] := 862.2261;
   DATA[2031,2] := 2.0;
   DATA[2031,3] := 2.0;
   DATA[2031,4] := 262.3686;
   DATA[2031,5] := 8.395155;
   DATA[2031,6] := 331.1971;
   DATA[2031,7] := 2.462179;
   DATA[2031,8] := 2.0;
   DATA[2031,9] := 2.0;
   DATA[2031,10] := 2.0;
   DATA[2031,11] := 19.76759;
   DATA[2031,12] := 2.209653;
   DATA[2031,13] := 801.7976;
   DATA[2031,14] := 1.0;
   DATA[2031,15] := 2.0;
   DATA[2031,16] := 1.0;
   DATA[2031,17] := 1.0;
   DATA[2031,18] := 1.0;
   DATA[2031,19] := 2.0;
   DATA[2031,20] := 148.808;
   DATA[2031,21] := 154.909;
   DATA[2031,22] := 1.718643;
   DATA[2031,23] := 831.0562;
   DATA[2031,24] := 2.0;
   DATA[2031,25] := 2.0;
   DATA[2031,26] := 7.874455;
   DATA[2031,27] := 143.9375;
   DATA[2031,28] := 262.1764;
   DATA[2031,29] := 12.07383;
   DATA[2031,30] := 1.726609;
   DATA[2031,31] := 1.291277;
   DATA[2031,32] := 0.7355248;
   DATA[2031,33] := 0.3084905;
   DATA[2031,34] := 2.0;
   DATA[2031,35] := 250.2243;
   DATA[2031,36] := 1.69801;
   DATA[2031,37] := 189.1823;
   DATA[2031,38] := 0.000128152;
   DATA[2031,39] := 1.0;
   DATA[2031,40] := 1.0;
   DATA[2032,0] := 2.508407;
   DATA[2032,1] := 862.5009;
   DATA[2032,2] := 2.0;
   DATA[2032,3] := 2.0;
   DATA[2032,4] := 262.3686;
   DATA[2032,5] := 8.395155;
   DATA[2032,6] := 331.1971;
   DATA[2032,7] := 2.462179;
   DATA[2032,8] := 2.0;
   DATA[2032,9] := 2.0;
   DATA[2032,10] := 2.0;
   DATA[2032,11] := 19.76759;
   DATA[2032,12] := 2.209653;
   DATA[2032,13] := 801.7976;
   DATA[2032,14] := 1.0;
   DATA[2032,15] := 2.0;
   DATA[2032,16] := 1.0;
   DATA[2032,17] := 1.0;
   DATA[2032,18] := 1.0;
   DATA[2032,19] := 2.0;
   DATA[2032,20] := 148.808;
   DATA[2032,21] := 154.909;
   DATA[2032,22] := 1.718643;
   DATA[2032,23] := 831.0177;
   DATA[2032,24] := 2.0;
   DATA[2032,25] := 2.0;
   DATA[2032,26] := 7.874455;
   DATA[2032,27] := 143.9375;
   DATA[2032,28] := 262.1764;
   DATA[2032,29] := 12.07383;
   DATA[2032,30] := 1.726609;
   DATA[2032,31] := 1.288715;
   DATA[2032,32] := 0.7355248;
   DATA[2032,33] := 0.3084905;
   DATA[2032,34] := 2.0;
   DATA[2032,35] := 250.2243;
   DATA[2032,36] := 1.69801;
   DATA[2032,37] := 189.1022;
   DATA[2032,38] := 0.000128152;
   DATA[2032,39] := 1.0;
   DATA[2032,40] := 1.0;
   DATA[2033,0] := 2.493034;
   DATA[2033,1] := 862.4616;
   DATA[2033,2] := 2.0;
   DATA[2033,3] := 2.0;
   DATA[2033,4] := 262.3686;
   DATA[2033,5] := 8.395155;
   DATA[2033,6] := 331.1971;
   DATA[2033,7] := 2.462179;
   DATA[2033,8] := 2.0;
   DATA[2033,9] := 2.0;
   DATA[2033,10] := 2.0;
   DATA[2033,11] := 19.76759;
   DATA[2033,12] := 2.209653;
   DATA[2033,13] := 801.3971;
   DATA[2033,14] := 1.0;
   DATA[2033,15] := 2.0;
   DATA[2033,16] := 1.0;
   DATA[2033,17] := 1.0;
   DATA[2033,18] := 1.0;
   DATA[2033,19] := 2.0;
   DATA[2033,20] := 148.808;
   DATA[2033,21] := 154.8834;
   DATA[2033,22] := 1.717361;
   DATA[2033,23] := 830.7485;
   DATA[2033,24] := 2.0;
   DATA[2033,25] := 2.0;
   DATA[2033,26] := 7.874455;
   DATA[2033,27] := 143.9375;
   DATA[2033,28] := 262.1764;
   DATA[2033,29] := 12.07383;
   DATA[2033,30] := 1.726609;
   DATA[2033,31] := 1.281798;
   DATA[2033,32] := 0.7355248;
   DATA[2033,33] := 0.3084905;
   DATA[2033,34] := 2.0;
   DATA[2033,35] := 250.2243;
   DATA[2033,36] := 1.69801;
   DATA[2033,37] := 189.0381;
   DATA[2033,38] := 0.000128152;
   DATA[2033,39] := 1.0;
   DATA[2033,40] := 1.0;
   DATA[2034,0] := 2.47702;
   DATA[2034,1] := 862.2653;
   DATA[2034,2] := 2.0;
   DATA[2034,3] := 2.0;
   DATA[2034,4] := 262.3686;
   DATA[2034,5] := 8.395155;
   DATA[2034,6] := 331.1971;
   DATA[2034,7] := 2.46282;
   DATA[2034,8] := 2.0;
   DATA[2034,9] := 2.0;
   DATA[2034,10] := 2.0;
   DATA[2034,11] := 19.74198;
   DATA[2034,12] := 2.208756;
   DATA[2034,13] := 801.6775;
   DATA[2034,14] := 1.0;
   DATA[2034,15] := 2.0;
   DATA[2034,16] := 1.0;
   DATA[2034,17] := 1.0;
   DATA[2034,18] := 1.0;
   DATA[2034,19] := 2.0;
   DATA[2034,20] := 148.808;
   DATA[2034,21] := 154.6783;
   DATA[2034,22] := 1.717361;
   DATA[2034,23] := 830.5947;
   DATA[2034,24] := 2.0;
   DATA[2034,25] := 2.0;
   DATA[2034,26] := 7.874455;
   DATA[2034,27] := 143.9375;
   DATA[2034,28] := 261.888;
   DATA[2034,29] := 12.07383;
   DATA[2034,30] := 1.725327;
   DATA[2034,31] := 1.277699;
   DATA[2034,32] := 0.7355248;
   DATA[2034,33] := 0.3084905;
   DATA[2034,34] := 2.0;
   DATA[2034,35] := 250.0641;
   DATA[2034,36] := 1.69801;
   DATA[2034,37] := 188.8779;
   DATA[2034,38] := 0.000128152;
   DATA[2034,39] := 1.0;
   DATA[2034,40] := 1.0;
   DATA[2035,0] := 2.456202;
   DATA[2035,1] := 862.1083;
   DATA[2035,2] := 2.0;
   DATA[2035,3] := 2.0;
   DATA[2035,4] := 262.3686;
   DATA[2035,5] := 8.395155;
   DATA[2035,6] := 331.1971;
   DATA[2035,7] := 2.46282;
   DATA[2035,8] := 2.0;
   DATA[2035,9] := 2.0;
   DATA[2035,10] := 2.0;
   DATA[2035,11] := 19.70997;
   DATA[2035,12] := 2.208756;
   DATA[2035,13] := 801.317;
   DATA[2035,14] := 1.0;
   DATA[2035,15] := 2.0;
   DATA[2035,16] := 1.0;
   DATA[2035,17] := 1.0;
   DATA[2035,18] := 1.0;
   DATA[2035,19] := 2.0;
   DATA[2035,20] := 148.808;
   DATA[2035,21] := 154.6783;
   DATA[2035,22] := 1.717361;
   DATA[2035,23] := 830.5563;
   DATA[2035,24] := 2.0;
   DATA[2035,25] := 2.0;
   DATA[2035,26] := 7.874455;
   DATA[2035,27] := 143.9375;
   DATA[2035,28] := 261.888;
   DATA[2035,29] := 12.07383;
   DATA[2035,30] := 1.723532;
   DATA[2035,31] := 1.260535;
   DATA[2035,32] := 0.7355248;
   DATA[2035,33] := 0.3084905;
   DATA[2035,34] := 2.0;
   DATA[2035,35] := 249.8558;
   DATA[2035,36] := 1.69801;
   DATA[2035,37] := 188.8138;
   DATA[2035,38] := 0.000128152;
   DATA[2035,39] := 1.0;
   DATA[2035,40] := 1.0;
   DATA[2036,0] := 2.445953;
   DATA[2036,1] := 862.2653;
   DATA[2036,2] := 2.0;
   DATA[2036,3] := 2.0;
   DATA[2036,4] := 262.3686;
   DATA[2036,5] := 8.395155;
   DATA[2036,6] := 331.1971;
   DATA[2036,7] := 2.463204;
   DATA[2036,8] := 2.0;
   DATA[2036,9] := 2.0;
   DATA[2036,10] := 2.0;
   DATA[2036,11] := 19.70997;
   DATA[2036,12] := 2.208756;
   DATA[2036,13] := 801.0767;
   DATA[2036,14] := 1.0;
   DATA[2036,15] := 2.0;
   DATA[2036,16] := 1.0;
   DATA[2036,17] := 1.0;
   DATA[2036,18] := 1.0;
   DATA[2036,19] := 2.0;
   DATA[2036,20] := 148.808;
   DATA[2036,21] := 154.6783;
   DATA[2036,22] := 1.716464;
   DATA[2036,23] := 831.1331;
   DATA[2036,24] := 2.0;
   DATA[2036,25] := 2.0;
   DATA[2036,26] := 7.874455;
   DATA[2036,27] := 143.9375;
   DATA[2036,28] := 261.888;
   DATA[2036,29] := 12.07383;
   DATA[2036,30] := 1.723532;
   DATA[2036,31] := 1.254259;
   DATA[2036,32] := 0.7355248;
   DATA[2036,33] := 0.3084905;
   DATA[2036,34] := 2.0;
   DATA[2036,35] := 249.8558;
   DATA[2036,36] := 1.69801;
   DATA[2036,37] := 188.8138;
   DATA[2036,38] := 0.000128152;
   DATA[2036,39] := 1.0;
   DATA[2036,40] := 1.0;
   DATA[2037,0] := 2.432822;
   DATA[2037,1] := 862.0691;
   DATA[2037,2] := 2.0;
   DATA[2037,3] := 2.0;
   DATA[2037,4] := 262.3686;
   DATA[2037,5] := 8.395155;
   DATA[2037,6] := 331.1971;
   DATA[2037,7] := 2.463589;
   DATA[2037,8] := 2.0;
   DATA[2037,9] := 2.0;
   DATA[2037,10] := 2.0;
   DATA[2037,11] := 19.75159;
   DATA[2037,12] := 2.208756;
   DATA[2037,13] := 801.1167;
   DATA[2037,14] := 1.0;
   DATA[2037,15] := 2.0;
   DATA[2037,16] := 1.0;
   DATA[2037,17] := 1.0;
   DATA[2037,18] := 1.0;
   DATA[2037,19] := 2.0;
   DATA[2037,20] := 148.808;
   DATA[2037,21] := 154.6783;
   DATA[2037,22] := 1.715824;
   DATA[2037,23] := 831.3253;
   DATA[2037,24] := 2.0;
   DATA[2037,25] := 2.0;
   DATA[2037,26] := 7.874455;
   DATA[2037,27] := 143.9375;
   DATA[2037,28] := 261.888;
   DATA[2037,29] := 12.07383;
   DATA[2037,30] := 1.723532;
   DATA[2037,31] := 1.241962;
   DATA[2037,32] := 0.7355248;
   DATA[2037,33] := 0.3077219;
   DATA[2037,34] := 2.0;
   DATA[2037,35] := 249.8558;
   DATA[2037,36] := 1.649953;
   DATA[2037,37] := 188.8138;
   DATA[2037,38] := 0.000128152;
   DATA[2037,39] := 1.0;
   DATA[2037,40] := 1.0;
   DATA[2038,0] := 2.432822;
   DATA[2038,1] := 862.0691;
   DATA[2038,2] := 2.0;
   DATA[2038,3] := 2.0;
   DATA[2038,4] := 262.3686;
   DATA[2038,5] := 8.395155;
   DATA[2038,6] := 331.1971;
   DATA[2038,7] := 2.463589;
   DATA[2038,8] := 2.0;
   DATA[2038,9] := 2.0;
   DATA[2038,10] := 2.0;
   DATA[2038,11] := 19.75159;
   DATA[2038,12] := 2.208756;
   DATA[2038,13] := 801.1167;
   DATA[2038,14] := 1.0;
   DATA[2038,15] := 2.0;
   DATA[2038,16] := 1.0;
   DATA[2038,17] := 1.0;
   DATA[2038,18] := 1.0;
   DATA[2038,19] := 2.0;
   DATA[2038,20] := 148.808;
   DATA[2038,21] := 154.6783;
   DATA[2038,22] := 1.715824;
   DATA[2038,23] := 831.3253;
   DATA[2038,24] := 2.0;
   DATA[2038,25] := 2.0;
   DATA[2038,26] := 7.874455;
   DATA[2038,27] := 143.9375;
   DATA[2038,28] := 261.888;
   DATA[2038,29] := 12.07383;
   DATA[2038,30] := 1.723532;
   DATA[2038,31] := 1.241962;
   DATA[2038,32] := 0.7355248;
   DATA[2038,33] := 0.3077219;
   DATA[2038,34] := 2.0;
   DATA[2038,35] := 249.8558;
   DATA[2038,36] := 1.649953;
   DATA[2038,37] := 188.8138;
   DATA[2038,38] := 0.000128152;
   DATA[2038,39] := 1.0;
   DATA[2038,40] := 1.0;
   DATA[2039,0] := 2.423213;
   DATA[2039,1] := 861.7158;
   DATA[2039,2] := 2.0;
   DATA[2039,3] := 2.0;
   DATA[2039,4] := 262.3686;
   DATA[2039,5] := 8.393232;
   DATA[2039,6] := 331.1971;
   DATA[2039,7] := 2.463589;
   DATA[2039,8] := 2.0;
   DATA[2039,9] := 2.0;
   DATA[2039,10] := 2.0;
   DATA[2039,11] := 19.77399;
   DATA[2039,12] := 2.210037;
   DATA[2039,13] := 800.9565;
   DATA[2039,14] := 1.0;
   DATA[2039,15] := 2.0;
   DATA[2039,16] := 1.0;
   DATA[2039,17] := 1.0;
   DATA[2039,18] := 1.0;
   DATA[2039,19] := 2.0;
   DATA[2039,20] := 148.808;
   DATA[2039,21] := 154.909;
   DATA[2039,22] := 1.715824;
   DATA[2039,23] := 831.3253;
   DATA[2039,24] := 2.0;
   DATA[2039,25] := 2.0;
   DATA[2039,26] := 7.874455;
   DATA[2039,27] := 143.9375;
   DATA[2039,28] := 261.888;
   DATA[2039,29] := 12.07383;
   DATA[2039,30] := 1.725455;
   DATA[2039,31] := 1.237351;
   DATA[2039,32] := 0.7355248;
   DATA[2039,33] := 0.3077219;
   DATA[2039,34] := 2.0;
   DATA[2039,35] := 250.032;
   DATA[2039,36] := 1.649953;
   DATA[2039,37] := 188.8138;
   DATA[2039,38] := 0.000128152;
   DATA[2039,39] := 1.0;
   DATA[2039,40] := 1.0;
   DATA[2040,0] := 2.423213;
   DATA[2040,1] := 862.0691;
   DATA[2040,2] := 2.0;
   DATA[2040,3] := 2.0;
   DATA[2040,4] := 262.3686;
   DATA[2040,5] := 8.393232;
   DATA[2040,6] := 331.1971;
   DATA[2040,7] := 2.463589;
   DATA[2040,8] := 2.0;
   DATA[2040,9] := 2.0;
   DATA[2040,10] := 2.0;
   DATA[2040,11] := 19.77399;
   DATA[2040,12] := 2.210037;
   DATA[2040,13] := 800.7562;
   DATA[2040,14] := 1.0;
   DATA[2040,15] := 2.0;
   DATA[2040,16] := 1.0;
   DATA[2040,17] := 1.0;
   DATA[2040,18] := 1.0;
   DATA[2040,19] := 2.0;
   DATA[2040,20] := 148.808;
   DATA[2040,21] := 155.0372;
   DATA[2040,22] := 1.715824;
   DATA[2040,23] := 831.556;
   DATA[2040,24] := 2.0;
   DATA[2040,25] := 2.0;
   DATA[2040,26] := 7.874455;
   DATA[2040,27] := 143.9375;
   DATA[2040,28] := 262.1764;
   DATA[2040,29] := 12.07383;
   DATA[2040,30] := 1.725583;
   DATA[2040,31] := 1.251953;
   DATA[2040,32] := 0.7355248;
   DATA[2040,33] := 0.3084905;
   DATA[2040,34] := 2.0;
   DATA[2040,35] := 250.0961;
   DATA[2040,36] := 1.649953;
   DATA[2040,37] := 188.9419;
   DATA[2040,38] := 0.000128152;
   DATA[2040,39] := 1.0;
   DATA[2040,40] := 1.0;
   DATA[2041,0] := 2.433783;
   DATA[2041,1] := 861.598;
   DATA[2041,2] := 2.0;
   DATA[2041,3] := 2.0;
   DATA[2041,4] := 262.3686;
   DATA[2041,5] := 8.393232;
   DATA[2041,6] := 331.0946;
   DATA[2041,7] := 2.463589;
   DATA[2041,8] := 2.0;
   DATA[2041,9] := 2.0;
   DATA[2041,10] := 2.0;
   DATA[2041,11] := 19.77399;
   DATA[2041,12] := 2.210037;
   DATA[2041,13] := 800.7162;
   DATA[2041,14] := 1.0;
   DATA[2041,15] := 2.0;
   DATA[2041,16] := 1.0;
   DATA[2041,17] := 1.0;
   DATA[2041,18] := 1.0;
   DATA[2041,19] := 2.0;
   DATA[2041,20] := 148.808;
   DATA[2041,21] := 155.0372;
   DATA[2041,22] := 1.718387;
   DATA[2041,23] := 831.5176;
   DATA[2041,24] := 2.0;
   DATA[2041,25] := 2.0;
   DATA[2041,26] := 7.874455;
   DATA[2041,27] := 143.9375;
   DATA[2041,28] := 262.1764;
   DATA[2041,29] := 12.07383;
   DATA[2041,30] := 1.726096;
   DATA[2041,31] := 1.267837;
   DATA[2041,32] := 0.7355248;
   DATA[2041,33] := 0.3084905;
   DATA[2041,34] := 2.0;
   DATA[2041,35] := 250.1923;
   DATA[2041,36] := 1.649953;
   DATA[2041,37] := 189.1342;
   DATA[2041,38] := 0.000128152;
   DATA[2041,39] := 1.0;
   DATA[2041,40] := 1.0;
   DATA[2042,0] := 2.487589;
   DATA[2042,1] := 861.6373;
   DATA[2042,2] := 2.0;
   DATA[2042,3] := 2.0;
   DATA[2042,4] := 262.3686;
   DATA[2042,5] := 8.393232;
   DATA[2042,6] := 331.0946;
   DATA[2042,7] := 2.463589;
   DATA[2042,8] := 2.0;
   DATA[2042,9] := 2.0;
   DATA[2042,10] := 2.0;
   DATA[2042,11] := 19.74198;
   DATA[2042,12] := 2.210037;
   DATA[2042,13] := 800.5159;
   DATA[2042,14] := 1.0;
   DATA[2042,15] := 2.0;
   DATA[2042,16] := 1.0;
   DATA[2042,17] := 1.0;
   DATA[2042,18] := 1.0;
   DATA[2042,19] := 2.0;
   DATA[2042,20] := 148.808;
   DATA[2042,21] := 154.8065;
   DATA[2042,22] := 1.718387;
   DATA[2042,23] := 831.7098;
   DATA[2042,24] := 2.0;
   DATA[2042,25] := 2.0;
   DATA[2042,26] := 7.874455;
   DATA[2042,27] := 143.9375;
   DATA[2042,28] := 262.1764;
   DATA[2042,29] := 12.07383;
   DATA[2042,30] := 1.728275;
   DATA[2042,31] := 1.280646;
   DATA[2042,32] := 0.7355248;
   DATA[2042,33] := 0.3070813;
   DATA[2042,34] := 2.0;
   DATA[2042,35] := 250.4005;
   DATA[2042,36] := 1.649953;
   DATA[2042,37] := 189.1662;
   DATA[2042,38] := 0.000128152;
   DATA[2042,39] := 1.0;
   DATA[2042,40] := 1.0;
   DATA[2043,0] := 2.531147;
   DATA[2043,1] := 861.3232;
   DATA[2043,2] := 2.0;
   DATA[2043,3] := 2.0;
   DATA[2043,4] := 262.3686;
   DATA[2043,5] := 8.393232;
   DATA[2043,6] := 331.0946;
   DATA[2043,7] := 2.461667;
   DATA[2043,8] := 2.0;
   DATA[2043,9] := 2.0;
   DATA[2043,10] := 2.0;
   DATA[2043,11] := 19.72598;
   DATA[2043,12] := 2.210037;
   DATA[2043,13] := 800.7162;
   DATA[2043,14] := 1.0;
   DATA[2043,15] := 2.0;
   DATA[2043,16] := 1.0;
   DATA[2043,17] := 1.0;
   DATA[2043,18] := 1.0;
   DATA[2043,19] := 2.0;
   DATA[2043,20] := 148.808;
   DATA[2043,21] := 154.8065;
   DATA[2043,22] := 1.718387;
   DATA[2043,23] := 831.556;
   DATA[2043,24] := 2.0;
   DATA[2043,25] := 2.0;
   DATA[2043,26] := 7.874455;
   DATA[2043,27] := 143.9375;
   DATA[2043,28] := 262.0802;
   DATA[2043,29] := 12.07383;
   DATA[2043,30] := 1.728275;
   DATA[2043,31] := 1.281798;
   DATA[2043,32] := 0.7355248;
   DATA[2043,33] := 0.3068251;
   DATA[2043,34] := 2.0;
   DATA[2043,35] := 250.4005;
   DATA[2043,36] := 1.649953;
   DATA[2043,37] := 189.1662;
   DATA[2043,38] := 0.000128152;
   DATA[2043,39] := 1.0;
   DATA[2043,40] := 1.0;
   DATA[2044,0] := 2.573744;
   DATA[2044,1] := 861.5195;
   DATA[2044,2] := 2.0;
   DATA[2044,3] := 2.0;
   DATA[2044,4] := 262.3686;
   DATA[2044,5] := 8.393232;
   DATA[2044,6] := 331.0946;
   DATA[2044,7] := 2.461667;
   DATA[2044,8] := 2.0;
   DATA[2044,9] := 2.0;
   DATA[2044,10] := 2.0;
   DATA[2044,11] := 19.72598;
   DATA[2044,12] := 2.210037;
   DATA[2044,13] := 800.5159;
   DATA[2044,14] := 1.0;
   DATA[2044,15] := 2.0;
   DATA[2044,16] := 1.0;
   DATA[2044,17] := 1.0;
   DATA[2044,18] := 1.0;
   DATA[2044,19] := 2.0;
   DATA[2044,20] := 148.808;
   DATA[2044,21] := 154.8065;
   DATA[2044,22] := 1.718387;
   DATA[2044,23] := 831.6329;
   DATA[2044,24] := 2.0;
   DATA[2044,25] := 2.0;
   DATA[2044,26] := 7.874455;
   DATA[2044,27] := 143.9375;
   DATA[2044,28] := 262.0802;
   DATA[2044,29] := 12.07383;
   DATA[2044,30] := 1.730069;
   DATA[2044,31] := 1.271935;
   DATA[2044,32] := 0.7355248;
   DATA[2044,33] := 0.3068251;
   DATA[2044,34] := 2.0;
   DATA[2044,35] := 250.4005;
   DATA[2044,36] := 1.746067;
   DATA[2044,37] := 189.2624;
   DATA[2044,38] := 0.000128152;
   DATA[2044,39] := 1.0;
   DATA[2044,40] := 1.0;
   DATA[2045,0] := 2.601928;
   DATA[2045,1] := 861.5195;
   DATA[2045,2] := 2.0;
   DATA[2045,3] := 2.0;
   DATA[2045,4] := 262.3686;
   DATA[2045,5] := 8.393232;
   DATA[2045,6] := 331.0946;
   DATA[2045,7] := 2.461667;
   DATA[2045,8] := 2.0;
   DATA[2045,9] := 2.0;
   DATA[2045,10] := 2.0;
   DATA[2045,11] := 19.72598;
   DATA[2045,12] := 2.210037;
   DATA[2045,13] := 800.3156;
   DATA[2045,14] := 1.0;
   DATA[2045,15] := 2.0;
   DATA[2045,16] := 1.0;
   DATA[2045,17] := 1.0;
   DATA[2045,18] := 1.0;
   DATA[2045,19] := 2.0;
   DATA[2045,20] := 148.808;
   DATA[2045,21] := 154.8065;
   DATA[2045,22] := 1.718387;
   DATA[2045,23] := 831.7867;
   DATA[2045,24] := 2.0;
   DATA[2045,25] := 2.0;
   DATA[2045,26] := 7.874455;
   DATA[2045,27] := 144.2451;
   DATA[2045,28] := 262.0802;
   DATA[2045,29] := 12.07383;
   DATA[2045,30] := 1.731351;
   DATA[2045,31] := 1.271935;
   DATA[2045,32] := 0.7355248;
   DATA[2045,33] := 0.3068251;
   DATA[2045,34] := 2.0;
   DATA[2045,35] := 250.5127;
   DATA[2045,36] := 1.762086;
   DATA[2045,37] := 189.2624;
   DATA[2045,38] := 0.000128152;
   DATA[2045,39] := 1.0;
   DATA[2045,40] := 1.0;
   DATA[2046,0] := 2.636198;
   DATA[2046,1] := 861.284;
   DATA[2046,2] := 2.0;
   DATA[2046,3] := 2.0;
   DATA[2046,4] := 262.3686;
   DATA[2046,5] := 8.393232;
   DATA[2046,6] := 331.0946;
   DATA[2046,7] := 2.461667;
   DATA[2046,8] := 2.0;
   DATA[2046,9] := 2.0;
   DATA[2046,10] := 2.0;
   DATA[2046,11] := 19.71957;
   DATA[2046,12] := 2.206963;
   DATA[2046,13] := 800.3958;
   DATA[2046,14] := 1.0;
   DATA[2046,15] := 2.0;
   DATA[2046,16] := 1.0;
   DATA[2046,17] := 1.0;
   DATA[2046,18] := 1.0;
   DATA[2046,19] := 2.0;
   DATA[2046,20] := 148.808;
   DATA[2046,21] := 154.8065;
   DATA[2046,22] := 1.718387;
   DATA[2046,23] := 832.3635;
   DATA[2046,24] := 2.0;
   DATA[2046,25] := 2.0;
   DATA[2046,26] := 7.874455;
   DATA[2046,27] := 144.2451;
   DATA[2046,28] := 262.0802;
   DATA[2046,29] := 12.07383;
   DATA[2046,30] := 1.731351;
   DATA[2046,31] := 1.271679;
   DATA[2046,32] := 0.7355248;
   DATA[2046,33] := 0.3068251;
   DATA[2046,34] := 2.0;
   DATA[2046,35] := 250.6409;
   DATA[2046,36] := 1.762086;
   DATA[2046,37] := 189.3585;
   DATA[2046,38] := 0.000128152;
   DATA[2046,39] := 1.0;
   DATA[2046,40] := 1.0;
   DATA[2047,0] := 2.653172;
   DATA[2047,1] := 861.441;
   DATA[2047,2] := 2.0;
   DATA[2047,3] := 2.0;
   DATA[2047,4] := 262.3686;
   DATA[2047,5] := 8.393232;
   DATA[2047,6] := 331.0946;
   DATA[2047,7] := 2.461667;
   DATA[2047,8] := 2.0;
   DATA[2047,9] := 2.0;
   DATA[2047,10] := 2.0;
   DATA[2047,11] := 19.71957;
   DATA[2047,12] := 2.206322;
   DATA[2047,13] := 800.3156;
   DATA[2047,14] := 1.0;
   DATA[2047,15] := 2.0;
   DATA[2047,16] := 1.0;
   DATA[2047,17] := 1.0;
   DATA[2047,18] := 1.0;
   DATA[2047,19] := 2.0;
   DATA[2047,20] := 148.808;
   DATA[2047,21] := 154.8065;
   DATA[2047,22] := 1.718387;
   DATA[2047,23] := 832.2866;
   DATA[2047,24] := 2.0;
   DATA[2047,25] := 2.0;
   DATA[2047,26] := 7.874455;
   DATA[2047,27] := 144.0913;
   DATA[2047,28] := 262.0802;
   DATA[2047,29] := 12.07383;
   DATA[2047,30] := 1.731351;
   DATA[2047,31] := 1.290637;
   DATA[2047,32] := 0.7355248;
   DATA[2047,33] := 0.3068251;
   DATA[2047,34] := 2.0;
   DATA[2047,35] := 250.6409;
   DATA[2047,36] := 1.681991;
   DATA[2047,37] := 189.4386;
   DATA[2047,38] := 0.000128152;
   DATA[2047,39] := 1.0;
   DATA[2047,40] := 1.0;
   DATA[2048,0] := 2.663421;
   DATA[2048,1] := 861.441;
   DATA[2048,2] := 2.0;
   DATA[2048,3] := 2.0;
   DATA[2048,4] := 262.3686;
   DATA[2048,5] := 8.393232;
   DATA[2048,6] := 331.0946;
   DATA[2048,7] := 2.461667;
   DATA[2048,8] := 2.0;
   DATA[2048,9] := 2.0;
   DATA[2048,10] := 2.0;
   DATA[2048,11] := 19.69396;
   DATA[2048,12] := 2.206322;
   DATA[2048,13] := 800.3156;
   DATA[2048,14] := 1.0;
   DATA[2048,15] := 2.0;
   DATA[2048,16] := 1.0;
   DATA[2048,17] := 1.0;
   DATA[2048,18] := 1.0;
   DATA[2048,19] := 2.0;
   DATA[2048,20] := 148.808;
   DATA[2048,21] := 155.0372;
   DATA[2048,22] := 1.718387;
   DATA[2048,23] := 832.3635;
   DATA[2048,24] := 2.0;
   DATA[2048,25] := 2.0;
   DATA[2048,26] := 7.874455;
   DATA[2048,27] := 143.8862;
   DATA[2048,28] := 262.0802;
   DATA[2048,29] := 12.07383;
   DATA[2048,30] := 1.731351;
   DATA[2048,31] := 1.291789;
   DATA[2048,32] := 0.7355248;
   DATA[2048,33] := 0.3063127;
   DATA[2048,34] := 2.0;
   DATA[2048,35] := 250.6248;
   DATA[2048,36] := 1.649953;
   DATA[2048,37] := 189.4386;
   DATA[2048,38] := 0.000128152;
   DATA[2048,39] := 1.0;
   DATA[2048,40] := 1.0;
   DATA[2049,0] := 2.664062;
   DATA[2049,1] := 861.284;
   DATA[2049,2] := 2.0;
   DATA[2049,3] := 2.0;
   DATA[2049,4] := 262.3686;
   DATA[2049,5] := 8.393232;
   DATA[2049,6] := 331.0946;
   DATA[2049,7] := 2.461667;
   DATA[2049,8] := 2.0;
   DATA[2049,9] := 2.0;
   DATA[2049,10] := 2.0;
   DATA[2049,11] := 19.67796;
   DATA[2049,12] := 2.206322;
   DATA[2049,13] := 800.596;
   DATA[2049,14] := 1.0;
   DATA[2049,15] := 2.0;
   DATA[2049,16] := 1.0;
   DATA[2049,17] := 1.0;
   DATA[2049,18] := 1.0;
   DATA[2049,19] := 2.0;
   DATA[2049,20] := 148.808;
   DATA[2049,21] := 155.0372;
   DATA[2049,22] := 1.715952;
   DATA[2049,23] := 832.9018;
   DATA[2049,24] := 2.0;
   DATA[2049,25] := 2.0;
   DATA[2049,26] := 7.874455;
   DATA[2049,27] := 143.8862;
   DATA[2049,28] := 262.0802;
   DATA[2049,29] := 12.07383;
   DATA[2049,30] := 1.730838;
   DATA[2049,31] := 1.291918;
   DATA[2049,32] := 0.7355248;
   DATA[2049,33] := 0.3063127;
   DATA[2049,34] := 2.0;
   DATA[2049,35] := 250.3525;
   DATA[2049,36] := 1.649953;
   DATA[2049,37] := 189.3265;
   DATA[2049,38] := 0.000128152;
   DATA[2049,39] := 1.0;
   DATA[2049,40] := 1.0;
   DATA[2050,0] := 2.628191;
   DATA[2050,1] := 861.6373;
   DATA[2050,2] := 2.0;
   DATA[2050,3] := 2.0;
   DATA[2050,4] := 262.3686;
   DATA[2050,5] := 8.393232;
   DATA[2050,6] := 331.0946;
   DATA[2050,7] := 2.463589;
   DATA[2050,8] := 2.0;
   DATA[2050,9] := 2.0;
   DATA[2050,10] := 2.0;
   DATA[2050,11] := 19.67796;
   DATA[2050,12] := 2.206322;
   DATA[2050,13] := 800.7162;
   DATA[2050,14] := 1.0;
   DATA[2050,15] := 2.0;
   DATA[2050,16] := 1.0;
   DATA[2050,17] := 1.0;
   DATA[2050,18] := 1.0;
   DATA[2050,19] := 2.0;
   DATA[2050,20] := 148.808;
   DATA[2050,21] := 155.0372;
   DATA[2050,22] := 1.715952;
   DATA[2050,23] := 832.7095;
   DATA[2050,24] := 2.0;
   DATA[2050,25] := 2.0;
   DATA[2050,26] := 7.874455;
   DATA[2050,27] := 143.8862;
   DATA[2050,28] := 262.0802;
   DATA[2050,29] := 12.07383;
   DATA[2050,30] := 1.728019;
   DATA[2050,31] := 1.286922;
   DATA[2050,32] := 0.7355248;
   DATA[2050,33] := 0.3063127;
   DATA[2050,34] := 2.0;
   DATA[2050,35] := 250.3525;
   DATA[2050,36] := 1.649953;
   DATA[2050,37] := 189.1823;
   DATA[2050,38] := 0.000128152;
   DATA[2050,39] := 1.0;
   DATA[2050,40] := 1.0;
   DATA[2051,0] := 2.620824;
   DATA[2051,1] := 861.441;
   DATA[2051,2] := 2.0;
   DATA[2051,3] := 2.0;
   DATA[2051,4] := 262.3686;
   DATA[2051,5] := 8.392271;
   DATA[2051,6] := 331.0946;
   DATA[2051,7] := 2.463589;
   DATA[2051,8] := 2.0;
   DATA[2051,9] := 2.0;
   DATA[2051,10] := 2.0;
   DATA[2051,11] := 19.67796;
   DATA[2051,12] := 2.206322;
   DATA[2051,13] := 800.7963;
   DATA[2051,14] := 1.0;
   DATA[2051,15] := 2.0;
   DATA[2051,16] := 1.0;
   DATA[2051,17] := 1.0;
   DATA[2051,18] := 1.0;
   DATA[2051,19] := 2.0;
   DATA[2051,20] := 148.808;
   DATA[2051,21] := 155.0372;
   DATA[2051,22] := 1.715952;
   DATA[2051,23] := 833.171;
   DATA[2051,24] := 2.0;
   DATA[2051,25] := 2.0;
   DATA[2051,26] := 7.874455;
   DATA[2051,27] := 143.8862;
   DATA[2051,28] := 262.0802;
   DATA[2051,29] := 12.07383;
   DATA[2051,30] := 1.726865;
   DATA[2051,31] := 1.280902;
   DATA[2051,32] := 0.7355248;
   DATA[2051,33] := 0.3063127;
   DATA[2051,34] := 2.0;
